C05448=1086.247,247.212,-78.817,176.012,22.627,153.611
C05449=1086.241,246.963,-78.790,176.009,22.624,153.611
C05450=1086.236,246.714,-78.763,176.007,22.621,153.611
C05451=1086.230,246.466,-78.736,176.004,22.619,153.611
C05452=1086.224,246.217,-78.710,176.002,22.616,153.610
C05453=1086.218,245.969,-78.683,175.999,22.613,153.610
C05454=1086.213,245.720,-78.656,175.996,22.610,153.610
C05455=1086.207,245.472,-78.629,175.994,22.607,153.610
C05456=1086.202,245.224,-78.603,175.991,22.604,153.610
C05457=1086.196,244.975,-78.576,175.988,22.602,153.609
C05458=1086.191,244.727,-78.549,175.985,22.598,153.609
C05459=1086.184,244.478,-78.522,175.982,22.596,153.609
C05460=1086.179,244.229,-78.495,175.980,22.593,153.608
C05461=1086.173,243.981,-78.468,175.977,22.590,153.608
C05462=1086.168,243.732,-78.441,175.974,22.587,153.608
C05463=1086.162,243.483,-78.415,175.972,22.584,153.608
C05464=1086.157,243.235,-78.389,175.969,22.581,153.608
C05465=1086.151,242.986,-78.362,175.967,22.578,153.607
C05466=1086.145,242.738,-78.335,175.964,22.576,153.607
C05467=1086.139,242.490,-78.309,175.961,22.573,153.607
C05468=1086.134,242.241,-78.282,175.958,22.570,153.607
C05469=1086.129,241.992,-78.255,175.955,22.567,153.607
C05470=1086.123,241.744,-78.229,175.953,22.564,153.606
C05471=1086.117,241.495,-78.202,175.950,22.561,153.606
C05472=1086.111,241.247,-78.176,175.947,22.558,153.606
C05473=1086.106,240.999,-78.149,175.945,22.556,153.606
C05474=1086.100,240.750,-78.123,175.942,22.553,153.605
C05475=1086.094,240.501,-78.096,175.939,22.550,153.605
C05476=1086.089,240.253,-78.070,175.936,22.547,153.605
C05477=1086.083,240.004,-78.044,175.934,22.544,153.605
C05478=1086.077,239.756,-78.017,175.931,22.542,153.604
C05479=1086.072,239.507,-77.990,175.928,22.538,153.604
C05480=1086.066,239.258,-77.964,175.926,22.536,153.604
C05481=1086.060,239.010,-77.938,175.923,22.533,153.604
C05482=1086.055,238.762,-77.911,175.921,22.530,153.604
C05483=1086.049,238.513,-77.885,175.918,22.527,153.603
C05484=1086.043,238.264,-77.859,175.915,22.525,153.603
C05485=1086.038,238.015,-77.833,175.912,22.522,153.603
C05486=1086.032,237.767,-77.806,175.909,22.519,153.603
C05487=1086.026,237.519,-77.779,175.907,22.516,153.602
C05488=1086.020,237.270,-77.754,175.904,22.513,153.602
C05489=1086.014,237.022,-77.727,175.902,22.511,153.602
C05490=1086.009,236.773,-77.701,175.899,22.507,153.602
C05491=1086.000,236.389,-77.661,175.895,22.503,153.601
C05492=1085.992,236.005,-77.620,175.891,22.498,153.601
C05493=1085.983,235.620,-77.580,175.887,22.495,153.601
C05494=1085.975,235.237,-77.539,175.882,22.490,153.601
C05495=1085.969,234.988,-77.513,175.880,22.487,153.600
C05496=1085.963,234.740,-77.487,175.877,22.484,153.600
C05497=1085.958,234.491,-77.461,175.875,22.482,153.600
C05498=1085.952,234.242,-77.435,175.872,22.479,153.600
C05499=1085.946,233.994,-77.409,175.869,22.476,153.599
C05500=1085.941,233.745,-77.383,175.867,22.473,153.599
C05501=1085.935,233.497,-77.357,175.864,22.470,153.599
C05502=1085.930,233.248,-77.331,175.861,22.467,153.599
C05503=1085.924,232.999,-77.305,175.858,22.464,153.598
C05504=1085.918,232.751,-77.279,175.856,22.462,153.598
C05505=1085.912,232.502,-77.253,175.853,22.459,153.598
C05506=1085.908,232.254,-77.227,175.851,22.456,153.598
C05507=1085.902,232.005,-77.201,175.848,22.453,153.598
C05508=1085.896,231.757,-77.175,175.846,22.451,153.597
C05509=1085.890,231.508,-77.149,175.843,22.447,153.597
C05510=1085.885,231.259,-77.123,175.840,22.445,153.597
C05511=1085.879,231.010,-77.097,175.837,22.442,153.597
C05512=1085.873,230.762,-77.072,175.835,22.440,153.596
C05513=1085.868,230.513,-77.046,175.832,22.436,153.596
C05514=1085.862,230.264,-77.020,175.829,22.434,153.596
C05515=1085.856,230.016,-76.994,175.827,22.431,153.596
C05516=1085.851,229.767,-76.969,175.824,22.428,153.596
C05517=1085.846,229.518,-76.943,175.822,22.425,153.595
C05518=1085.839,229.270,-76.917,175.819,22.422,153.595
C05519=1085.834,229.021,-76.891,175.816,22.420,153.595
C05520=1085.828,228.773,-76.866,175.813,22.417,153.595
C05521=1085.822,228.524,-76.840,175.811,22.414,153.594
C05522=1085.817,228.276,-76.815,175.808,22.411,153.594
C05523=1085.811,228.027,-76.789,175.806,22.408,153.594
C05524=1085.806,227.778,-76.763,175.803,22.406,153.594
C05525=1085.799,227.529,-76.738,175.801,22.403,153.594
C05526=1085.795,227.281,-76.712,175.798,22.400,153.594
C05527=1085.788,227.032,-76.687,175.795,22.397,153.593
C05528=1085.783,226.783,-76.661,175.792,22.395,153.593
C05529=1085.777,226.535,-76.635,175.790,22.392,153.593
C05530=1085.772,226.286,-76.610,175.787,22.389,153.593
C05531=1085.766,226.038,-76.584,175.785,22.386,153.592
C05532=1085.760,225.789,-76.559,175.782,22.383,153.592
C05533=1085.754,225.541,-76.534,175.780,22.381,153.592
C05534=1085.749,225.292,-76.508,175.777,22.378,153.592
C05535=1085.743,225.043,-76.482,175.775,22.375,153.591
C05536=1085.737,224.794,-76.456,175.772,22.373,153.591
C05537=1085.732,224.546,-76.431,175.769,22.369,153.591
C05538=1085.726,224.297,-76.405,175.767,22.367,153.591
C05539=1085.720,224.048,-76.380,175.764,22.364,153.591
C05540=1085.716,223.800,-76.355,175.762,22.362,153.590
C05541=1085.709,223.551,-76.330,175.759,22.358,153.590
C05542=1085.704,223.302,-76.304,175.757,22.356,153.590
C05543=1085.695,222.910,-76.264,175.752,22.351,153.590
C05544=1085.686,222.517,-76.225,175.748,22.347,153.589
C05545=1085.677,222.124,-76.184,175.744,22.342,153.589
C05546=1085.669,221.732,-76.144,175.740,22.338,153.589
C05547=1085.663,221.483,-76.119,175.737,22.335,153.588
C05548=1085.657,221.235,-76.094,175.735,22.333,153.588
C05549=1085.651,220.986,-76.069,175.732,22.329,153.588
C05550=1085.646,220.737,-76.043,175.730,22.327,153.588
C05551=1085.640,220.488,-76.019,175.727,22.324,153.588
C05552=1085.634,220.240,-75.994,175.724,22.321,153.587
C05553=1085.629,219.992,-75.969,175.722,22.319,153.587
C05554=1085.623,219.742,-75.943,175.719,22.316,153.587
C05555=1085.617,219.493,-75.918,175.717,22.314,153.587
C05556=1085.612,219.246,-75.893,175.714,22.310,153.587
C05557=1085.606,218.996,-75.868,175.712,22.308,153.586
C05558=1085.601,218.748,-75.843,175.709,22.305,153.586
C05559=1085.595,218.499,-75.818,175.706,22.302,153.586
C05560=1085.589,218.250,-75.793,175.704,22.299,153.586
C05561=1085.583,218.002,-75.768,175.701,22.297,153.586
C05562=1085.578,217.752,-75.743,175.699,22.294,153.585
C05563=1085.572,217.504,-75.718,175.696,22.291,153.585
C05564=1085.567,217.255,-75.693,175.694,22.288,153.585
C05565=1085.561,217.007,-75.668,175.691,22.286,153.585
C05566=1085.555,216.758,-75.644,175.689,22.283,153.584
C05567=1085.550,216.510,-75.618,175.686,22.280,153.584
C05568=1085.544,216.260,-75.593,175.684,22.277,153.584
C05569=1085.539,216.012,-75.568,175.681,22.275,153.584
C05570=1085.533,215.763,-75.544,175.678,22.272,153.584
C05571=1085.527,215.515,-75.519,175.676,22.269,153.583
C05572=1085.521,215.266,-75.494,175.673,22.266,153.583
C05573=1085.516,215.018,-75.469,175.671,22.264,153.583
C05574=1085.510,214.768,-75.444,175.668,22.260,153.583
C05575=1085.505,214.520,-75.420,175.666,22.258,153.583
C05576=1085.499,214.271,-75.394,175.663,22.255,153.582
C05577=1085.494,214.022,-75.370,175.660,22.252,153.582
C05578=1085.487,213.774,-75.345,175.658,22.250,153.582
C05579=1085.483,213.525,-75.320,175.655,22.247,153.582
C05580=1085.477,213.276,-75.295,175.653,22.244,153.581
C05581=1085.471,213.028,-75.270,175.650,22.241,153.581
C05582=1085.465,212.778,-75.246,175.648,22.238,153.581
C05583=1085.460,212.530,-75.222,175.646,22.236,153.581
C05584=1085.455,212.281,-75.197,175.643,22.233,153.581
C05585=1085.449,212.032,-75.172,175.640,22.231,153.580
C05586=1085.443,211.784,-75.148,175.637,22.227,153.580
C05587=1085.437,211.535,-75.123,175.635,22.225,153.580
C05588=1085.432,211.286,-75.099,175.633,22.222,153.580
C05589=1085.426,211.037,-75.073,175.630,22.219,153.580
C05590=1085.421,210.789,-75.049,175.628,22.216,153.579
C05591=1085.415,210.540,-75.025,175.625,22.214,153.579
C05592=1085.409,210.291,-75.000,175.622,22.211,153.579
C05593=1085.404,210.042,-74.976,175.620,22.209,153.579
C05594=1085.398,209.794,-74.951,175.617,22.206,153.579
C05595=1085.388,209.405,-74.913,175.614,22.202,153.578
C05596=1085.380,209.017,-74.875,175.610,22.197,153.578
C05597=1085.372,208.628,-74.837,175.605,22.193,153.578
C05598=1085.363,208.239,-74.799,175.602,22.188,153.577
C05599=1085.339,207.211,-74.700,175.519,22.146,153.580
C05600=1085.334,206.963,-74.676,175.517,22.144,153.580
C05601=1085.329,206.714,-74.652,175.514,22.142,153.580
C05602=1085.322,206.465,-74.628,175.511,22.140,153.580
C05603=1085.317,206.216,-74.604,175.509,22.138,153.580
C05604=1085.312,205.967,-74.580,175.506,22.136,153.580
C05605=1085.306,205.718,-74.557,175.504,22.135,153.580
C05606=1085.301,205.470,-74.533,175.501,22.133,153.580
C05607=1085.295,205.221,-74.508,175.498,22.131,153.580
C05608=1085.289,204.972,-74.485,175.495,22.129,153.580
C05609=1085.284,204.723,-74.461,175.493,22.127,153.580
C05610=1085.278,204.475,-74.437,175.490,22.125,153.580
C05611=1085.273,204.226,-74.414,175.488,22.123,153.580
C05612=1085.267,203.977,-74.389,175.485,22.122,153.580
C05613=1085.262,203.728,-74.366,175.483,22.120,153.580
C05614=1085.256,203.480,-74.342,175.479,22.118,153.580
C05615=1085.251,203.230,-74.317,175.477,22.116,153.580
C05616=1085.245,202.981,-74.295,175.475,22.114,153.580
C05617=1085.239,202.733,-74.270,175.472,22.112,153.580
C05618=1085.234,202.484,-74.247,175.470,22.111,153.580
C05619=1085.228,202.235,-74.223,175.467,22.109,153.580
C05620=1085.223,201.986,-74.200,175.465,22.107,153.580
C05621=1085.217,201.738,-74.176,175.462,22.106,153.580
C05622=1085.211,201.488,-74.153,175.459,22.103,153.580
C05623=1085.205,201.240,-74.129,175.456,22.102,153.581
C05624=1085.199,200.991,-74.106,175.454,22.100,153.581
C05625=1085.194,200.742,-74.082,175.451,22.098,153.580
C05626=1085.188,200.494,-74.059,175.449,22.096,153.580
C05627=1085.183,200.245,-74.034,175.446,22.095,153.581
C05628=1085.177,199.996,-74.012,175.444,22.093,153.581
C05629=1085.171,199.746,-73.988,175.441,22.091,153.581
C05630=1085.166,199.498,-73.964,175.439,22.090,153.581
C05631=1085.160,199.249,-73.941,175.435,22.088,153.581
C05632=1085.154,199.001,-73.917,175.433,22.086,153.581
C05633=1085.149,198.752,-73.894,175.430,22.084,153.581
C05634=1085.143,198.503,-73.871,175.428,22.082,153.581
C05635=1085.137,198.254,-73.847,175.426,22.081,153.581
C05636=1085.132,198.005,-73.824,175.423,22.079,153.581
C05637=1085.126,197.756,-73.801,175.420,22.077,153.581
C05638=1085.120,197.508,-73.777,175.418,22.076,153.581
C05639=1085.115,197.259,-73.754,175.416,22.074,153.581
C05640=1085.110,197.010,-73.731,175.413,22.072,153.581
C05641=1085.104,196.762,-73.707,175.410,22.070,153.581
C05642=1085.098,196.513,-73.684,175.407,22.068,153.581
C05643=1085.093,196.263,-73.660,175.405,22.066,153.581
C05644=1085.087,196.015,-73.638,175.402,22.065,153.581
C05645=1085.081,195.765,-73.614,175.400,22.063,153.581
C05646=1085.076,195.516,-73.590,175.397,22.061,153.581
C05647=1085.070,195.267,-73.567,175.395,22.060,153.581
C05648=1085.064,195.019,-73.544,175.392,22.058,153.581
C05649=1085.058,194.770,-73.521,175.390,22.056,153.581
C05650=1085.054,194.521,-73.498,175.387,22.054,153.581
C05651=1085.048,194.273,-73.474,175.385,22.052,153.581
C05652=1085.042,194.024,-73.451,175.382,22.050,153.581
C05653=1085.036,193.775,-73.428,175.380,22.049,153.581
C05654=1085.031,193.526,-73.405,175.377,22.047,153.581
C05655=1085.026,193.277,-73.382,175.375,22.045,153.581
C05656=1085.020,193.028,-73.359,175.372,22.043,153.581
C05657=1085.014,192.779,-73.336,175.369,22.041,153.581
C05658=1085.009,192.531,-73.312,175.367,22.039,153.581
C05659=1085.003,192.282,-73.289,175.364,22.038,153.581
C05660=1084.997,192.003,-73.264,175.362,22.036,153.581
C05661=1084.990,191.725,-73.238,175.358,22.033,153.581
C05662=1084.985,191.447,-73.211,175.356,22.032,153.581
C05663=1084.978,191.168,-73.187,175.354,22.030,153.581
C05664=1084.973,190.919,-73.163,175.351,22.028,153.581
C05665=1084.968,190.670,-73.140,175.349,22.026,153.581
C05666=1084.962,190.421,-73.117,175.346,22.024,153.581
C05667=1084.956,190.172,-73.094,175.344,22.022,153.581
C05668=1084.950,189.923,-73.071,175.340,22.021,153.581
C05669=1084.946,189.675,-73.048,175.338,22.019,153.581
C05670=1084.940,189.426,-73.025,175.335,22.017,153.581
C05671=1084.935,189.177,-73.002,175.333,22.015,153.581
C05672=1084.929,188.928,-72.979,175.330,22.013,153.581
C05673=1084.923,188.679,-72.956,175.328,22.011,153.581
C05674=1084.917,188.430,-72.933,175.326,22.010,153.581
C05675=1084.913,188.182,-72.910,175.323,22.008,153.581
C05676=1084.907,187.933,-72.887,175.321,22.006,153.581
C05677=1084.902,187.684,-72.864,175.318,22.004,153.581
C05678=1084.896,187.435,-72.841,175.316,22.002,153.581
C05679=1084.890,187.186,-72.819,175.313,22.000,153.581
C05680=1084.885,186.937,-72.796,175.311,21.999,153.581
C05681=1084.879,186.689,-72.774,175.308,21.997,153.581
C05682=1084.874,186.439,-72.750,175.306,21.995,153.581
C05683=1084.869,186.190,-72.727,175.304,21.993,153.581
C05684=1084.863,185.941,-72.705,175.301,21.991,153.581
C05685=1084.858,185.693,-72.682,175.299,21.989,153.580
C05686=1084.852,185.444,-72.659,175.296,21.988,153.580
C05687=1084.847,185.195,-72.636,175.294,21.986,153.580
C05688=1084.841,184.946,-72.613,175.291,21.984,153.580
C05689=1084.836,184.697,-72.591,175.289,21.982,153.580
C05690=1084.830,184.448,-72.568,175.286,21.981,153.581
C05691=1084.824,184.200,-72.546,175.284,21.979,153.581
C05692=1084.818,183.951,-72.523,175.281,21.977,153.581
C05693=1084.813,183.701,-72.501,175.279,21.975,153.580
C05694=1084.807,183.452,-72.478,175.276,21.974,153.581
C05695=1084.801,183.204,-72.456,175.274,21.972,153.581
C05696=1084.795,182.954,-72.434,175.271,21.970,153.581
C05697=1084.789,182.705,-72.411,175.269,21.968,153.581
C05698=1084.784,182.457,-72.388,175.266,21.966,153.581
C05699=1084.778,182.208,-72.366,175.264,21.965,153.581
C05700=1084.772,181.959,-72.343,175.261,21.963,153.581
C05701=1084.767,181.710,-72.321,175.259,21.961,153.581
C05702=1084.761,181.461,-72.298,175.257,21.960,153.581
C05703=1084.755,181.212,-72.276,175.255,21.958,153.581
C05704=1084.750,180.963,-72.254,175.252,21.957,153.581
C05705=1084.744,180.714,-72.231,175.250,21.955,153.581
C05706=1084.739,180.465,-72.209,175.247,21.953,153.581
C05707=1084.732,180.216,-72.187,175.245,21.951,153.581
C05708=1084.727,179.967,-72.164,175.243,21.950,153.581
C05709=1084.722,179.719,-72.142,175.240,21.948,153.581
C05710=1084.715,179.470,-72.119,175.238,21.946,153.581
C05711=1084.710,179.221,-72.097,175.235,21.944,153.581
C05712=1084.704,178.972,-72.074,175.233,21.943,153.581
C05713=1084.699,178.723,-72.053,175.230,21.941,153.581
C05714=1084.693,178.474,-72.030,175.228,21.939,153.581
C05715=1084.687,178.225,-72.008,175.225,21.937,153.581
C05716=1084.681,177.975,-71.986,175.223,21.935,153.581
C05717=1084.676,177.727,-71.964,175.220,21.933,153.581
C05718=1084.671,177.478,-71.941,175.218,21.932,153.581
C05719=1084.664,177.229,-71.919,175.215,21.930,153.581
C05720=1084.659,176.980,-71.897,175.213,21.928,153.581
C05721=1084.654,176.731,-71.874,175.210,21.927,153.581
C05722=1084.648,176.482,-71.853,175.209,21.925,153.581
C05723=1084.642,176.233,-71.830,175.206,21.923,153.581
C05724=1084.636,175.954,-71.806,175.203,21.921,153.581
C05725=1084.630,175.676,-71.781,175.201,21.919,153.581
C05726=1084.623,175.398,-71.756,175.198,21.917,153.581
C05727=1084.617,175.119,-71.731,175.196,21.916,153.581
C05728=1084.612,174.870,-71.709,175.193,21.914,153.581
C05729=1084.606,174.620,-71.687,175.191,21.912,153.581
C05730=1084.600,174.372,-71.665,175.188,21.910,153.581
C05731=1084.595,174.123,-71.642,175.186,21.908,153.581
C05732=1084.589,173.874,-71.621,175.183,21.906,153.581
C05733=1084.584,173.625,-71.599,175.181,21.904,153.580
C05734=1084.578,173.376,-71.576,175.179,21.903,153.580
C05735=1084.573,173.127,-71.555,175.176,21.901,153.580
C05736=1084.567,172.878,-71.532,175.174,21.899,153.580
C05737=1084.561,172.629,-71.511,175.171,21.897,153.580
C05738=1084.556,172.380,-71.488,175.169,21.895,153.580
C05739=1084.550,172.131,-71.467,175.167,21.894,153.580
C05740=1084.545,171.882,-71.445,175.165,21.892,153.580
C05741=1084.539,171.633,-71.423,175.162,21.890,153.580
C05742=1084.533,171.384,-71.401,175.160,21.888,153.580
C05743=1084.528,171.136,-71.378,175.158,21.886,153.580
C05744=1084.522,170.886,-71.357,175.155,21.885,153.580
C05745=1084.517,170.637,-71.335,175.153,21.883,153.580
C05746=1084.511,170.388,-71.313,175.150,21.881,153.580
C05747=1084.506,170.139,-71.291,175.148,21.879,153.580
C05748=1084.500,169.890,-71.270,175.146,21.878,153.580
C05749=1084.495,169.641,-71.247,175.144,21.876,153.580
C05750=1084.489,169.392,-71.226,175.141,21.874,153.580
C05751=1084.483,169.143,-71.203,175.139,21.872,153.580
C05752=1084.478,168.895,-71.181,175.136,21.870,153.580
C05753=1084.472,168.645,-71.160,175.134,21.868,153.580
C05754=1084.467,168.397,-71.138,175.132,21.866,153.580
C05755=1084.461,168.147,-71.116,175.129,21.864,153.580
C05756=1084.457,167.898,-71.094,175.127,21.862,153.580
C05757=1084.450,167.649,-71.073,175.125,21.861,153.580
C05758=1084.446,167.400,-71.051,175.123,21.859,153.580
C05759=1084.439,167.151,-71.029,175.120,21.857,153.580
C05760=1084.435,166.902,-71.007,175.118,21.855,153.580
C05761=1084.428,166.653,-70.986,175.116,21.854,153.580
C05762=1084.424,166.404,-70.964,175.113,21.852,153.580
C05763=1084.418,166.156,-70.943,175.111,21.849,153.580
C05764=1084.412,165.907,-70.921,175.109,21.848,153.580
C05765=1084.407,165.658,-70.899,175.107,21.846,153.580
C05766=1084.401,165.409,-70.877,175.104,21.844,153.580
C05767=1084.396,165.160,-70.856,175.102,21.842,153.580
C05768=1084.390,164.910,-70.835,175.100,21.841,153.580
C05769=1084.385,164.661,-70.813,175.097,21.839,153.580
C05770=1084.380,164.413,-70.792,175.095,21.836,153.579
C05771=1084.374,164.163,-70.769,175.093,21.835,153.579
C05772=1084.369,163.915,-70.748,175.091,21.833,153.579
C05773=1084.363,163.665,-70.726,175.088,21.831,153.579
C05774=1084.358,163.417,-70.705,175.086,21.830,153.579
C05775=1084.353,163.168,-70.684,175.084,21.828,153.579
C05776=1084.347,162.918,-70.662,175.081,21.825,153.579
C05777=1084.342,162.670,-70.641,175.079,21.823,153.579
C05778=1084.336,162.420,-70.618,175.077,21.822,153.579
C05779=1084.331,162.172,-70.597,175.075,21.820,153.579
C05780=1084.326,161.923,-70.575,175.072,21.818,153.579
C05781=1084.320,161.673,-70.554,175.070,21.816,153.579
C05782=1084.314,161.424,-70.533,175.068,21.814,153.579
C05783=1084.308,161.175,-70.511,175.065,21.812,153.579
C05784=1084.303,160.926,-70.489,175.064,21.811,153.579
C05785=1084.298,160.677,-70.469,175.061,21.809,153.579
C05786=1084.292,160.428,-70.447,175.059,21.807,153.579
C05787=1084.286,160.180,-70.426,175.056,21.805,153.579
C05788=1084.280,159.901,-70.402,175.054,21.804,153.579
C05789=1084.273,159.621,-70.378,175.052,21.801,153.579
C05790=1084.267,159.342,-70.354,175.049,21.799,153.579
C05791=1084.261,159.062,-70.331,175.046,21.797,153.579
C05792=1084.256,158.814,-70.309,175.044,21.796,153.579
C05793=1084.250,158.565,-70.288,175.042,21.794,153.579
C05794=1084.244,158.316,-70.267,175.040,21.792,153.579
C05795=1084.239,158.067,-70.246,175.037,21.790,153.579
C05796=1084.233,157.818,-70.224,175.035,21.788,153.578
C05797=1084.227,157.569,-70.204,175.033,21.786,153.578
C05798=1084.222,157.320,-70.182,175.031,21.784,153.578
C05799=1084.217,157.070,-70.161,175.028,21.783,153.578
C05800=1084.211,156.822,-70.140,175.026,21.781,153.578
C05801=1084.206,156.573,-70.118,175.024,21.779,153.578
C05802=1084.200,156.323,-70.097,175.022,21.777,153.578
C05803=1084.194,156.075,-70.076,175.020,21.775,153.578
C05804=1084.189,155.826,-70.056,175.017,21.773,153.578
C05805=1084.183,155.577,-70.034,175.015,21.771,153.578
C05806=1084.178,155.327,-70.013,175.012,21.770,153.578
C05807=1084.172,155.079,-69.992,175.011,21.768,153.578
C05808=1084.166,154.829,-69.971,175.008,21.766,153.578
C05809=1084.161,154.581,-69.950,175.006,21.764,153.578
C05810=1084.155,154.331,-69.929,175.004,21.763,153.578
C05811=1084.149,154.082,-69.908,175.001,21.760,153.578
C05812=1084.144,153.833,-69.887,175.000,21.759,153.578
C05813=1084.138,153.585,-69.866,174.997,21.757,153.578
C05814=1084.132,153.335,-69.845,174.995,21.755,153.578
C05815=1084.127,153.086,-69.824,174.993,21.753,153.578
C05816=1084.122,152.837,-69.803,174.991,21.752,153.578
C05817=1084.116,152.587,-69.782,174.989,21.750,153.578
C05818=1084.110,152.339,-69.761,174.986,21.748,153.578
C05819=1084.105,152.090,-69.740,174.984,21.746,153.578
C05820=1084.099,151.841,-69.719,174.981,21.744,153.578
C05821=1084.094,151.591,-69.698,174.980,21.743,153.578
C05822=1084.088,151.342,-69.678,174.978,21.740,153.577
C05823=1084.082,151.094,-69.657,174.975,21.738,153.577
C05824=1084.076,150.844,-69.636,174.973,21.737,153.577
C05825=1084.071,150.595,-69.616,174.971,21.735,153.577
C05826=1084.065,150.347,-69.594,174.969,21.733,153.577
C05827=1084.060,150.097,-69.574,174.967,21.731,153.577
C05828=1084.054,149.848,-69.553,174.964,21.729,153.577
C05829=1084.049,149.599,-69.532,174.963,21.728,153.577
C05830=1084.043,149.350,-69.511,174.960,21.726,153.577
C05831=1084.038,149.101,-69.490,174.958,21.723,153.577
C05832=1084.032,148.851,-69.470,174.955,21.722,153.577
C05833=1084.026,148.603,-69.449,174.954,21.720,153.577
C05834=1084.021,148.354,-69.428,174.951,21.718,153.577
C05835=1084.015,148.105,-69.408,174.949,21.716,153.577
C05836=1084.010,147.856,-69.387,174.947,21.714,153.577
C05837=1084.003,147.607,-69.366,174.945,21.713,153.577
C05838=1083.998,147.357,-69.346,174.943,21.711,153.577
C05839=1083.993,147.108,-69.325,174.940,21.709,153.577
C05840=1083.988,146.859,-69.305,174.938,21.707,153.577
C05841=1083.981,146.610,-69.284,174.937,21.705,153.576
C05842=1083.975,146.361,-69.263,174.934,21.703,153.576
C05843=1083.970,146.112,-69.242,174.932,21.701,153.576
C05844=1083.965,145.863,-69.222,174.929,21.700,153.576
C05845=1083.959,145.614,-69.202,174.928,21.698,153.576
C05846=1083.953,145.364,-69.181,174.925,21.696,153.576
C05847=1083.948,145.115,-69.160,174.923,21.694,153.576
C05848=1083.942,144.866,-69.140,174.921,21.692,153.576
C05849=1083.937,144.617,-69.120,174.919,21.690,153.576
C05850=1083.931,144.369,-69.099,174.917,21.688,153.576
C05851=1083.924,144.119,-69.078,174.914,21.687,153.576
C05852=1083.919,143.840,-69.055,174.912,21.685,153.576
C05853=1083.913,143.561,-69.032,174.910,21.682,153.576
C05854=1083.906,143.282,-69.010,174.907,21.680,153.576
C05855=1083.900,143.002,-68.987,174.905,21.678,153.576
C05856=1083.895,142.753,-68.966,174.903,21.676,153.576
C05857=1083.889,142.503,-68.945,174.901,21.675,153.576
C05858=1083.883,142.255,-68.926,174.899,21.672,153.576
C05859=1083.878,142.005,-68.905,174.896,21.671,153.576
C05860=1083.872,141.756,-68.884,174.894,21.669,153.576
C05861=1083.866,141.508,-68.864,174.893,21.667,153.575
C05862=1083.861,141.258,-68.844,174.890,21.665,153.575
C05863=1083.855,141.010,-68.824,174.888,21.663,153.575
C05864=1083.850,140.760,-68.803,174.886,21.661,153.575
C05865=1083.845,140.511,-68.783,174.884,21.659,153.575
C05866=1083.838,140.262,-68.762,174.882,21.657,153.575
C05867=1083.833,140.013,-68.742,174.879,21.655,153.575
C05868=1083.827,139.764,-68.722,174.878,21.654,153.575
C05869=1083.822,139.515,-68.701,174.875,21.652,153.575
C05870=1083.816,139.265,-68.682,174.873,21.649,153.575
C05871=1083.811,139.016,-68.662,174.872,21.648,153.575
C05872=1083.805,138.767,-68.641,174.869,21.646,153.575
C05873=1083.799,138.518,-68.621,174.867,21.644,153.575
C05874=1083.794,138.269,-68.601,174.865,21.642,153.575
C05875=1083.788,138.020,-68.581,174.863,21.641,153.575
C05876=1083.783,137.771,-68.560,174.861,21.638,153.574
C05877=1083.777,137.521,-68.540,174.858,21.636,153.574
C05878=1083.771,137.272,-68.520,174.857,21.635,153.574
C05879=1083.765,137.023,-68.500,174.854,21.633,153.574
C05880=1083.759,136.774,-68.480,174.852,21.631,153.574
C05881=1083.754,136.525,-68.459,174.850,21.629,153.574
C05882=1083.748,136.276,-68.440,174.848,21.627,153.574
C05883=1083.743,136.027,-68.420,174.846,21.625,153.574
C05884=1083.737,135.778,-68.400,174.844,21.624,153.574
C05885=1083.732,135.529,-68.379,174.842,21.621,153.574
C05886=1083.726,135.279,-68.360,174.840,21.619,153.574
C05887=1083.720,135.030,-68.340,174.838,21.618,153.574
C05888=1083.715,134.781,-68.319,174.836,21.616,153.574
C05889=1083.709,134.533,-68.299,174.833,21.614,153.574
C05890=1083.704,134.283,-68.280,174.832,21.612,153.573
C05891=1083.698,134.034,-68.260,174.830,21.610,153.573
C05892=1083.693,133.785,-68.239,174.827,21.608,153.573
C05893=1083.687,133.535,-68.220,174.826,21.606,153.573
C05894=1083.681,133.287,-68.200,174.823,21.604,153.573
C05895=1083.676,133.038,-68.179,174.821,21.602,153.573
C05896=1083.670,132.788,-68.160,174.820,21.601,153.573
C05897=1083.665,132.539,-68.139,174.817,21.599,153.573
C05898=1083.659,132.290,-68.120,174.815,21.596,153.573
C05899=1083.653,132.041,-68.100,174.813,21.595,153.573
C05900=1083.647,131.792,-68.080,174.811,21.593,153.573
C05901=1083.642,131.542,-68.060,174.809,21.591,153.573
C05902=1083.636,131.293,-68.041,174.807,21.589,153.573
C05903=1083.631,131.044,-68.021,174.805,21.587,153.572
C05904=1083.625,130.795,-68.001,174.803,21.585,153.572
C05905=1083.619,130.546,-67.981,174.801,21.584,153.572
C05906=1083.614,130.297,-67.962,174.799,21.581,153.572
C05907=1083.608,130.048,-67.942,174.796,21.579,153.572
C05908=1083.602,129.798,-67.922,174.795,21.578,153.572
C05909=1083.596,129.549,-67.902,174.793,21.576,153.572
C05910=1083.590,129.300,-67.883,174.790,21.574,153.572
C05911=1083.584,129.051,-67.863,174.789,21.572,153.572
C05912=1083.579,128.801,-67.843,174.786,21.570,153.572
C05913=1083.573,128.553,-67.823,174.784,21.568,153.572
C05914=1083.568,128.303,-67.804,174.783,21.566,153.572
C05915=1083.562,128.054,-67.784,174.780,21.564,153.572
C05916=1083.556,127.774,-67.762,174.778,21.562,153.572
C05917=1083.548,127.495,-67.740,174.776,21.560,153.572
C05918=1083.543,127.216,-67.718,174.773,21.558,153.571
C05919=1083.536,126.937,-67.697,174.771,21.555,153.571
C05920=1083.531,126.687,-67.676,174.770,21.554,153.571
C05921=1083.525,126.438,-67.657,174.767,21.552,153.571
C05922=1083.519,126.189,-67.637,174.765,21.550,153.571
C05923=1083.513,125.940,-67.618,174.763,21.548,153.571
C05924=1083.508,125.690,-67.599,174.761,21.546,153.571
C05925=1083.502,125.442,-67.579,174.760,21.545,153.571
C05926=1083.497,125.193,-67.560,174.757,21.542,153.571
C05927=1083.491,124.943,-67.540,174.755,21.540,153.571
C05928=1083.485,124.695,-67.520,174.754,21.538,153.571
C05929=1083.480,124.445,-67.501,174.751,21.536,153.571
C05930=1083.474,124.195,-67.481,174.749,21.534,153.570
C05931=1083.468,123.947,-67.461,174.747,21.533,153.570
C05932=1083.463,123.697,-67.442,174.745,21.530,153.570
C05933=1083.457,123.448,-67.423,174.744,21.529,153.570
C05934=1083.452,123.200,-67.403,174.741,21.527,153.570
C05935=1083.446,122.950,-67.384,174.739,21.525,153.570
C05936=1083.440,122.701,-67.365,174.738,21.523,153.570
C05937=1083.435,122.451,-67.346,174.735,21.521,153.570
C05938=1083.429,122.203,-67.326,174.733,21.518,153.570
C05939=1083.423,121.953,-67.306,174.731,21.517,153.570
C05940=1083.418,121.704,-67.288,174.729,21.515,153.570
C05941=1083.412,121.455,-67.268,174.728,21.513,153.569
C05942=1083.406,121.205,-67.249,174.725,21.511,153.569
C05943=1083.400,120.957,-67.229,174.723,21.509,153.569
C05944=1083.395,120.707,-67.209,174.722,21.507,153.569
C05945=1083.390,120.458,-67.190,174.719,21.505,153.569
C05946=1083.385,120.209,-67.171,174.718,21.503,153.569
C05947=1083.379,119.959,-67.152,174.716,21.501,153.569
C05948=1083.373,119.711,-67.132,174.713,21.499,153.569
C05949=1083.367,119.461,-67.113,174.712,21.497,153.569
C05950=1083.362,119.212,-67.094,174.710,21.495,153.568
C05951=1083.357,118.963,-67.075,174.708,21.493,153.568
C05952=1083.351,118.713,-67.055,174.706,21.491,153.568
C05953=1083.345,118.464,-67.036,174.704,21.489,153.568
C05954=1083.340,118.215,-67.017,174.702,21.487,153.568
C05955=1083.334,117.966,-66.998,174.700,21.485,153.568
C05956=1083.329,117.716,-66.979,174.699,21.483,153.568
C05957=1083.323,117.468,-66.959,174.696,21.481,153.568
C05958=1083.318,117.219,-66.940,174.694,21.479,153.568
C05959=1083.312,116.969,-66.921,174.693,21.477,153.567
C05960=1083.306,116.720,-66.901,174.690,21.475,153.567
C05961=1083.301,116.471,-66.883,174.689,21.473,153.567
C05962=1083.295,116.222,-66.863,174.687,21.470,153.567
C05963=1083.290,115.972,-66.844,174.684,21.469,153.567
C05964=1083.284,115.723,-66.825,174.683,21.467,153.567
C05965=1083.279,115.474,-66.806,174.681,21.464,153.567
C05966=1083.273,115.225,-66.787,174.679,21.463,153.567
C05967=1083.268,114.975,-66.767,174.677,21.461,153.567
C05968=1083.262,114.727,-66.749,174.675,21.459,153.566
C05969=1083.256,114.478,-66.730,174.673,21.456,153.566
C05970=1083.250,114.228,-66.711,174.671,21.454,153.566
C05971=1083.245,113.979,-66.692,174.669,21.452,153.566
C05972=1083.240,113.729,-66.673,174.667,21.451,153.566
C05973=1083.234,113.480,-66.654,174.666,21.449,153.566
C05974=1083.228,113.231,-66.635,174.663,21.446,153.566
C05975=1083.223,112.982,-66.616,174.662,21.445,153.566
C05976=1083.217,112.733,-66.597,174.660,21.442,153.566
C05977=1083.211,112.483,-66.578,174.658,21.440,153.565
C05978=1083.206,112.235,-66.560,174.656,21.439,153.565
C05979=1083.200,111.985,-66.540,174.654,21.436,153.565
C05980=1083.195,111.754,-66.523,174.652,21.435,153.565
C05981=1083.190,111.524,-66.505,174.651,21.433,153.565
C05982=1083.184,111.293,-66.488,174.649,21.430,153.565
C05983=1083.179,111.062,-66.471,174.647,21.429,153.565
C05984=1083.174,110.832,-66.453,174.645,21.427,153.565
C05985=1083.169,110.601,-66.436,174.643,21.425,153.565
C05986=1083.163,110.370,-66.419,174.642,21.423,153.565
C05987=1083.158,110.141,-66.401,174.640,21.421,153.565
C05988=1083.152,109.891,-66.382,174.638,21.420,153.564
C05989=1083.147,109.641,-66.364,174.636,21.418,153.564
C05990=1083.140,109.392,-66.345,174.634,21.416,153.564
C05991=1083.135,109.143,-66.326,174.632,21.413,153.564
C05992=1083.130,108.894,-66.307,174.631,21.412,153.564
C05993=1083.123,108.645,-66.288,174.628,21.410,153.564
C05994=1083.118,108.396,-66.270,174.626,21.407,153.564
C05995=1083.113,108.146,-66.251,174.625,21.406,153.564
C05996=1083.107,107.898,-66.233,174.623,21.403,153.564
C05997=1083.101,107.648,-66.214,174.621,21.401,153.563
C05998=1083.095,107.399,-66.195,174.619,21.400,153.563
C05999=1083.090,107.150,-66.177,174.617,21.398,153.563
C06000=1083.084,106.900,-66.157,174.615,21.395,153.563
C06001=1083.078,106.651,-66.139,174.614,21.393,153.563
C06002=1083.073,106.402,-66.120,174.611,21.391,153.563
C06003=1083.067,106.153,-66.102,174.610,21.389,153.563
C06004=1083.062,105.903,-66.084,174.608,21.387,153.563
C06005=1083.056,105.654,-66.064,174.606,21.385,153.562
C06006=1083.050,105.404,-66.046,174.604,21.383,153.562
C06007=1083.045,105.156,-66.028,174.602,21.381,153.562
C06008=1083.038,104.906,-66.009,174.601,21.379,153.562
C06009=1083.034,104.657,-65.991,174.598,21.377,153.562
C06010=1083.027,104.408,-65.972,174.597,21.375,153.562
C06011=1083.022,104.159,-65.953,174.595,21.373,153.562
C06012=1083.017,103.909,-65.935,174.593,21.371,153.562
C06013=1083.010,103.660,-65.916,174.591,21.368,153.561
C06014=1083.006,103.411,-65.898,174.590,21.367,153.561
C06015=1082.999,103.162,-65.879,174.587,21.365,153.561
C06016=1082.993,102.845,-65.856,174.585,21.362,153.561
C06017=1082.986,102.528,-65.833,174.583,21.359,153.561
C06018=1082.978,102.212,-65.809,174.580,21.356,153.561
C06019=1082.971,101.895,-65.785,174.578,21.354,153.561
C06020=1082.966,101.645,-65.767,174.576,21.352,153.560
C06021=1082.960,101.396,-65.749,174.574,21.350,153.560
C06022=1082.955,101.147,-65.730,174.573,21.348,153.560
C06023=1082.949,100.898,-65.712,174.571,21.345,153.560
C06024=1082.942,100.648,-65.694,174.569,21.344,153.560
C06025=1082.937,100.399,-65.675,174.567,21.342,153.560
C06026=1082.931,100.150,-65.657,174.566,21.340,153.560
C06027=1082.925,99.901,-65.639,174.563,21.337,153.559
C06028=1082.920,99.651,-65.620,174.562,21.336,153.559
C06029=1082.915,99.402,-65.603,174.560,21.333,153.559
C06030=1082.908,99.153,-65.584,174.558,21.332,153.559
C06031=1082.903,98.904,-65.566,174.556,21.329,153.559
C06032=1082.897,98.655,-65.547,174.555,21.328,153.559
C06033=1082.891,98.405,-65.530,174.552,21.325,153.559
C06034=1082.886,98.155,-65.511,174.551,21.323,153.559
C06035=1082.880,97.907,-65.493,174.549,21.321,153.558
C06036=1082.874,97.657,-65.475,174.547,21.319,153.558
C06037=1082.869,97.407,-65.456,174.545,21.317,153.558
C06038=1082.863,97.159,-65.438,174.544,21.315,153.558
C06039=1082.857,96.910,-65.420,174.541,21.313,153.558
C06040=1082.852,96.660,-65.402,174.539,21.310,153.558
C06041=1082.846,96.411,-65.384,174.538,21.308,153.558
C06042=1082.840,96.162,-65.366,174.536,21.306,153.557
C06043=1082.835,95.912,-65.348,174.534,21.305,153.557
C06044=1082.828,95.634,-65.327,174.532,21.302,153.557
C06045=1082.822,95.353,-65.306,174.530,21.299,153.557
C06046=1082.815,95.074,-65.287,174.529,21.297,153.557
C06047=1082.809,94.795,-65.266,174.526,21.295,153.557
C06048=1082.804,94.545,-65.249,174.524,21.293,153.557
C06049=1082.797,94.296,-65.230,174.523,21.291,153.557
C06050=1082.792,94.047,-65.212,174.520,21.289,153.556
C06051=1082.787,93.798,-65.194,174.519,21.287,153.556
C06052=1082.781,93.548,-65.176,174.517,21.284,153.556
C06053=1082.776,93.299,-65.158,174.516,21.283,153.556
C06054=1082.769,93.050,-65.139,174.513,21.280,153.556
C06055=1082.764,92.801,-65.122,174.512,21.278,153.556
C06056=1082.758,92.552,-65.104,174.510,21.276,153.555
C06057=1082.753,92.302,-65.086,174.509,21.274,153.555
C06058=1082.748,92.053,-65.068,174.506,21.271,153.555
C06059=1082.741,91.803,-65.050,174.505,21.270,153.555
C06060=1082.736,91.554,-65.032,174.503,21.268,153.555
C06061=1082.731,91.305,-65.014,174.501,21.266,153.555
C06062=1082.725,91.055,-64.996,174.499,21.263,153.555
C06063=1082.719,90.806,-64.978,174.498,21.261,153.554
C06064=1082.713,90.557,-64.960,174.496,21.259,153.554
C06065=1082.708,90.308,-64.943,174.494,21.257,153.554
C06066=1082.702,90.058,-64.925,174.493,21.255,153.554
C06067=1082.696,89.809,-64.907,174.491,21.253,153.554
C06068=1082.690,89.560,-64.889,174.489,21.251,153.554
C06069=1082.684,89.311,-64.871,174.487,21.249,153.554
C06070=1082.678,89.062,-64.854,174.486,21.247,153.554
C06071=1082.672,88.812,-64.836,174.483,21.244,153.553
C06072=1082.667,88.563,-64.818,174.482,21.243,153.553
C06073=1082.661,88.314,-64.800,174.480,21.240,153.553
C06074=1082.655,88.064,-64.783,174.478,21.238,153.553
C06075=1082.650,87.815,-64.765,174.476,21.236,153.553
C06076=1082.644,87.566,-64.747,174.475,21.234,153.553
C06077=1082.639,87.316,-64.729,174.473,21.232,153.553
C06078=1082.633,87.067,-64.711,174.471,21.230,153.552
C06079=1082.627,86.817,-64.693,174.469,21.228,153.552
C06080=1082.622,86.568,-64.676,174.468,21.226,153.552
C06081=1082.616,86.319,-64.658,174.465,21.223,153.552
C06082=1082.610,86.069,-64.640,174.464,21.221,153.552
C06083=1082.604,85.820,-64.623,174.463,21.219,153.552
C06084=1082.599,85.571,-64.605,174.461,21.217,153.551
C06085=1082.593,85.321,-64.587,174.459,21.215,153.551
C06086=1082.588,85.072,-64.570,174.457,21.213,153.551
C06087=1082.582,84.823,-64.553,174.456,21.211,153.551
C06088=1082.576,84.573,-64.535,174.454,21.208,153.551
C06089=1082.570,84.324,-64.517,174.452,21.206,153.551
C06090=1082.564,84.075,-64.500,174.450,21.204,153.551
C06091=1082.559,83.826,-64.483,174.449,21.202,153.550
C06092=1082.553,83.576,-64.465,174.446,21.200,153.550
C06093=1082.547,83.327,-64.447,174.445,21.198,153.550
C06094=1082.541,83.078,-64.430,174.444,21.196,153.550
C06095=1082.536,82.828,-64.413,174.441,21.194,153.550
C06096=1082.530,82.579,-64.395,174.440,21.192,153.550
C06097=1082.525,82.330,-64.377,174.438,21.189,153.550
C06098=1082.519,82.081,-64.360,174.437,21.188,153.549
C06099=1082.513,81.831,-64.342,174.434,21.185,153.549
C06100=1082.508,81.581,-64.325,174.433,21.183,153.549
C06101=1082.502,81.332,-64.307,174.431,21.180,153.549
C06102=1082.497,81.083,-64.290,174.430,21.178,153.549
C06103=1082.491,80.834,-64.272,174.427,21.176,153.548
C06104=1082.485,80.585,-64.254,174.426,21.174,153.548
C06105=1082.480,80.335,-64.238,174.425,21.172,153.548
C06106=1082.474,80.086,-64.220,174.423,21.170,153.548
C06107=1082.468,79.836,-64.202,174.421,21.168,153.548
C06108=1082.462,79.557,-64.183,174.419,21.165,153.548
C06109=1082.456,79.278,-64.164,174.417,21.163,153.548
C06110=1082.449,78.999,-64.144,174.416,21.160,153.547
C06111=1082.443,78.719,-64.125,174.414,21.158,153.547
C06112=1082.437,78.470,-64.107,174.411,21.156,153.547
C06113=1082.432,78.221,-64.090,174.410,21.154,153.547
C06114=1082.426,77.971,-64.073,174.408,21.151,153.547
C06115=1082.420,77.722,-64.056,174.407,21.149,153.546
C06116=1082.414,77.472,-64.038,174.405,21.147,153.546
C06117=1082.409,77.223,-64.021,174.403,21.145,153.546
C06118=1082.403,76.974,-64.004,174.402,21.143,153.546
C06119=1082.397,76.725,-63.986,174.399,21.141,153.546
C06120=1082.391,76.475,-63.969,174.398,21.139,153.546
C06121=1082.386,76.226,-63.952,174.396,21.136,153.546
C06122=1082.380,75.976,-63.935,174.395,21.134,153.545
C06123=1082.374,75.727,-63.918,174.393,21.132,153.545
C06124=1082.369,75.478,-63.900,174.391,21.130,153.545
C06125=1082.362,75.228,-63.884,174.390,21.128,153.545
C06126=1082.357,74.979,-63.866,174.388,21.126,153.545
C06127=1082.352,74.729,-63.849,174.386,21.124,153.545
C06128=1082.346,74.480,-63.832,174.384,21.121,153.544
C06129=1082.340,74.232,-63.815,174.383,21.119,153.544
C06130=1082.334,73.981,-63.797,174.381,21.117,153.544
C06131=1082.328,73.732,-63.780,174.379,21.115,153.544
C06132=1082.322,73.483,-63.764,174.378,21.113,153.544
C06133=1082.317,73.234,-63.746,174.376,21.111,153.544
C06134=1082.312,72.984,-63.729,174.375,21.108,153.543
C06135=1082.305,72.736,-63.712,174.373,21.106,153.543
C06136=1082.300,72.486,-63.695,174.371,21.104,153.543
C06137=1082.294,72.236,-63.677,174.370,21.102,153.543
C06138=1082.288,71.987,-63.661,174.368,21.099,153.543
C06139=1082.283,71.738,-63.644,174.366,21.097,153.543
C06140=1082.277,71.488,-63.627,174.364,21.095,153.542
C06141=1082.271,71.239,-63.610,174.363,21.093,153.542
C06142=1082.266,70.990,-63.593,174.361,21.091,153.542
C06143=1082.261,70.740,-63.576,174.359,21.089,153.542
C06144=1082.255,70.491,-63.559,174.358,21.087,153.542
C06145=1082.249,70.241,-63.542,174.356,21.084,153.541
C06146=1082.242,69.992,-63.525,174.355,21.082,153.541
C06147=1082.237,69.743,-63.508,174.353,21.080,153.541
C06148=1082.232,69.493,-63.491,174.351,21.077,153.541
C06149=1082.226,69.244,-63.474,174.350,21.075,153.541
C06150=1082.221,68.995,-63.457,174.348,21.073,153.541
C06151=1082.214,68.746,-63.440,174.346,21.071,153.540
C06152=1082.209,68.496,-63.424,174.345,21.069,153.540
C06153=1082.203,68.246,-63.407,174.343,21.067,153.540
C06154=1082.197,67.997,-63.389,174.341,21.065,153.540
C06155=1082.191,67.748,-63.373,174.339,21.062,153.540
C06156=1082.186,67.498,-63.356,174.338,21.060,153.540
C06157=1082.180,67.249,-63.339,174.337,21.058,153.539
C06158=1082.174,67.000,-63.322,174.335,21.056,153.539
C06159=1082.168,66.750,-63.306,174.333,21.054,153.539
C06160=1082.163,66.501,-63.289,174.331,21.051,153.539
C06161=1082.157,66.252,-63.272,174.330,21.049,153.539
C06162=1082.152,66.002,-63.256,174.328,21.047,153.539
C06163=1082.146,65.753,-63.239,174.326,21.045,153.538
C06164=1082.140,65.504,-63.222,174.325,21.043,153.538
C06165=1082.134,65.255,-63.205,174.323,21.040,153.538
C06166=1082.128,65.004,-63.189,174.322,21.038,153.538
C06167=1082.123,64.755,-63.172,174.320,21.036,153.538
C06168=1082.116,64.506,-63.155,174.318,21.034,153.538
C06169=1082.111,64.256,-63.138,174.317,21.032,153.537
C06170=1082.105,64.007,-63.122,174.315,21.029,153.537
C06171=1082.099,63.758,-63.106,174.313,21.027,153.537
C06172=1082.093,63.478,-63.087,174.311,21.025,153.537
C06173=1082.086,63.199,-63.068,174.310,21.022,153.537
C06174=1082.079,62.919,-63.050,174.308,21.020,153.536
C06175=1082.073,62.640,-63.031,174.306,21.018,153.536
C06176=1082.067,62.391,-63.015,174.304,21.016,153.536
C06177=1082.061,62.142,-62.998,174.303,21.014,153.536
C06178=1082.055,61.892,-62.981,174.301,21.011,153.536
C06179=1082.049,61.643,-62.965,174.299,21.009,153.536
C06180=1082.044,61.393,-62.948,174.297,21.006,153.535
C06181=1082.038,61.144,-62.932,174.296,21.004,153.535
C06182=1082.032,60.894,-62.915,174.295,21.002,153.535
C06183=1082.026,60.645,-62.899,174.293,21.000,153.535
C06184=1082.020,60.395,-62.883,174.291,20.998,153.535
C06185=1082.015,60.146,-62.866,174.290,20.996,153.535
C06186=1082.009,59.897,-62.849,174.288,20.994,153.534
C06187=1082.003,59.648,-62.833,174.286,20.992,153.534
C06188=1081.997,59.398,-62.816,174.284,20.989,153.534
C06189=1081.991,59.149,-62.800,174.283,20.987,153.534
C06190=1081.985,58.900,-62.784,174.282,20.985,153.534
C06191=1081.980,58.650,-62.767,174.280,20.982,153.533
C06192=1081.974,58.401,-62.751,174.278,20.980,153.533
C06193=1081.968,58.151,-62.734,174.277,20.979,153.533
C06194=1081.962,57.902,-62.718,174.275,20.976,153.533
C06195=1081.956,57.653,-62.702,174.274,20.974,153.533
C06196=1081.951,57.403,-62.685,174.271,20.972,153.533
C06197=1081.945,57.154,-62.669,174.270,20.970,153.533
C06198=1081.939,56.904,-62.653,174.269,20.967,153.532
C06199=1081.933,56.655,-62.636,174.267,20.965,153.532
C06200=1081.927,56.406,-62.620,174.265,20.963,153.532
C06201=1081.922,56.156,-62.603,174.264,20.961,153.532
C06202=1081.916,55.907,-62.587,174.262,20.959,153.532
C06203=1081.910,55.657,-62.571,174.261,20.957,153.531
C06204=1081.904,55.408,-62.554,174.259,20.954,153.531
C06205=1081.899,55.159,-62.539,174.257,20.952,153.531
C06206=1081.893,54.909,-62.523,174.256,20.950,153.531
C06207=1081.888,54.660,-62.506,174.254,20.947,153.531
C06208=1081.882,54.410,-62.490,174.252,20.945,153.531
C06209=1081.876,54.161,-62.474,174.251,20.943,153.530
C06210=1081.870,53.912,-62.457,174.249,20.940,153.530
C06211=1081.864,53.662,-62.441,174.248,20.938,153.530
C06212=1081.858,53.413,-62.425,174.247,20.937,153.530
C06213=1081.852,53.164,-62.409,174.244,20.934,153.530
C06214=1081.847,52.913,-62.393,174.243,20.932,153.529
C06215=1081.841,52.664,-62.376,174.241,20.929,153.529
C06216=1081.836,52.415,-62.360,174.240,20.927,153.529
C06217=1081.830,52.166,-62.344,174.238,20.925,153.529
C06218=1081.824,51.917,-62.328,174.236,20.923,153.529
C06219=1081.818,51.667,-62.312,174.235,20.920,153.528
C06220=1081.812,51.417,-62.296,174.234,20.918,153.528
C06221=1081.807,51.168,-62.280,174.232,20.916,153.528
C06222=1081.801,50.918,-62.263,174.230,20.914,153.528
C06223=1081.796,50.670,-62.247,174.229,20.912,153.528
C06224=1081.790,50.420,-62.232,174.227,20.909,153.527
C06225=1081.784,50.170,-62.215,174.226,20.907,153.527
C06226=1081.778,49.921,-62.199,174.224,20.905,153.527
C06227=1081.772,49.672,-62.183,174.222,20.903,153.527
C06228=1081.767,49.422,-62.167,174.221,20.900,153.527
C06229=1081.761,49.173,-62.151,174.220,20.898,153.526
C06230=1081.756,48.924,-62.135,174.218,20.896,153.526
C06231=1081.750,48.674,-62.119,174.217,20.893,153.526
C06232=1081.744,48.424,-62.103,174.214,20.891,153.526
C06233=1081.739,48.175,-62.086,174.213,20.889,153.526
C06234=1081.733,47.926,-62.071,174.212,20.887,153.526
C06235=1081.728,47.676,-62.055,174.210,20.884,153.525
C06236=1081.721,47.396,-62.036,174.208,20.882,153.525
C06237=1081.714,47.117,-62.019,174.207,20.879,153.525
C06238=1081.708,46.838,-62.002,174.205,20.877,153.525
C06239=1081.702,46.557,-61.983,174.203,20.874,153.524
C06240=1081.696,46.308,-61.967,174.202,20.872,153.524
C06241=1081.691,46.059,-61.951,174.200,20.870,153.524
C06242=1081.685,45.809,-61.936,174.199,20.867,153.524
C06243=1081.679,45.560,-61.919,174.197,20.865,153.524
C06244=1081.673,45.310,-61.903,174.195,20.863,153.523
C06245=1081.668,45.061,-61.888,174.194,20.860,153.523
C06246=1081.662,44.812,-61.872,174.193,20.859,153.523
C06247=1081.657,44.562,-61.856,174.191,20.856,153.523
C06248=1081.651,44.312,-61.840,174.189,20.854,153.523
C06249=1081.646,44.063,-61.825,174.188,20.852,153.522
C06250=1081.640,43.814,-61.808,174.186,20.849,153.522
C06251=1081.634,43.565,-61.792,174.185,20.847,153.522
C06252=1081.628,43.315,-61.777,174.184,20.845,153.522
C06253=1081.623,43.066,-61.761,174.181,20.842,153.522
C06254=1081.616,42.816,-61.746,174.180,20.840,153.521
C06255=1081.610,42.567,-61.730,174.179,20.838,153.521
C06256=1081.605,42.317,-61.714,174.177,20.835,153.521
C06257=1081.599,42.068,-61.698,174.176,20.833,153.521
C06258=1081.594,41.818,-61.683,174.174,20.832,153.521
C06259=1081.588,41.569,-61.666,174.172,20.829,153.521
C06260=1081.582,41.319,-61.651,174.171,20.827,153.520
C06261=1081.576,41.071,-61.636,174.170,20.825,153.520
C06262=1081.570,40.821,-61.620,174.167,20.822,153.520
C06263=1081.565,40.571,-61.604,174.166,20.820,153.520
C06264=1081.559,40.322,-61.589,174.165,20.818,153.519
C06265=1081.554,40.072,-61.573,174.163,20.815,153.519
C06266=1081.547,39.823,-61.557,174.162,20.813,153.519
C06267=1081.541,39.573,-61.542,174.160,20.811,153.519
C06268=1081.536,39.324,-61.526,174.158,20.808,153.519
C06269=1081.530,39.074,-61.510,174.157,20.806,153.519
C06270=1081.525,38.825,-61.495,174.156,20.804,153.518
C06271=1081.519,38.576,-61.479,174.154,20.802,153.518
C06272=1081.513,38.326,-61.464,174.152,20.800,153.518
C06273=1081.507,38.076,-61.448,174.151,20.798,153.518
C06274=1081.502,37.828,-61.433,174.149,20.795,153.517
C06275=1081.496,37.578,-61.418,174.148,20.793,153.517
C06276=1081.490,37.329,-61.401,174.147,20.791,153.517
C06277=1081.484,37.079,-61.386,174.144,20.788,153.517
C06278=1081.478,36.830,-61.371,174.143,20.786,153.517
C06279=1081.472,36.580,-61.355,174.142,20.784,153.516
C06280=1081.467,36.330,-61.339,174.141,20.782,153.516
C06281=1081.461,36.081,-61.325,174.138,20.779,153.516
C06282=1081.455,35.831,-61.309,174.137,20.777,153.516
C06283=1081.449,35.582,-61.293,174.136,20.775,153.516
C06284=1081.443,35.332,-61.278,174.134,20.773,153.516
C06285=1081.438,35.083,-61.263,174.133,20.771,153.515
C06286=1081.432,34.834,-61.247,174.131,20.769,153.515
C06287=1081.426,34.584,-61.232,174.129,20.766,153.515
C06288=1081.421,34.335,-61.217,174.128,20.764,153.515
C06289=1081.414,34.085,-61.202,174.127,20.762,153.515
C06290=1081.408,33.836,-61.185,174.125,20.759,153.514
C06291=1081.403,33.587,-61.170,174.123,20.757,153.514
C06292=1081.397,33.337,-61.155,174.122,20.755,153.514
C06293=1081.391,33.087,-61.140,174.121,20.753,153.514
C06294=1081.385,32.838,-61.125,174.119,20.750,153.514
C06295=1081.379,32.589,-61.109,174.118,20.748,153.513
C06296=1081.374,32.339,-61.094,174.116,20.746,153.513
C06297=1081.368,32.090,-61.079,174.114,20.743,153.513
C06298=1081.362,31.840,-61.063,174.113,20.741,153.513
C06299=1081.357,31.591,-61.049,174.112,20.739,153.513
C06300=1081.350,31.311,-61.031,174.110,20.737,153.512
C06301=1081.344,31.031,-61.013,174.108,20.734,153.512
C06302=1081.337,30.752,-60.997,174.106,20.732,153.512
C06303=1081.331,30.472,-60.980,174.104,20.729,153.512
C06304=1081.325,30.223,-60.964,174.103,20.727,153.512
C06305=1081.319,29.974,-60.949,174.102,20.724,153.511
C06306=1081.313,29.724,-60.934,174.101,20.722,153.511
C06307=1081.308,29.475,-60.919,174.098,20.720,153.511
C06308=1081.302,29.225,-60.903,174.097,20.717,153.511
C06309=1081.296,28.976,-60.889,174.096,20.715,153.510
C06310=1081.290,28.726,-60.873,174.094,20.713,153.510
C06311=1081.285,28.477,-60.859,174.093,20.711,153.510
C06312=1081.279,28.227,-60.843,174.091,20.708,153.510
C06313=1081.273,27.977,-60.828,174.089,20.706,153.510
C06314=1081.268,27.728,-60.813,174.088,20.704,153.510
C06315=1081.261,27.478,-60.798,174.087,20.702,153.509
C06316=1081.255,27.229,-60.784,174.086,20.700,153.509
C06317=1081.250,26.979,-60.768,174.083,20.697,153.509
C06318=1081.243,26.730,-60.753,174.082,20.695,153.509
C06319=1081.238,26.481,-60.738,174.081,20.693,153.509
C06320=1081.232,26.231,-60.723,174.079,20.690,153.508
C06321=1081.226,25.982,-60.708,174.078,20.688,153.508
C06322=1081.221,25.732,-60.693,174.076,20.686,153.508
C06323=1081.215,25.483,-60.678,174.075,20.684,153.508
C06324=1081.209,25.233,-60.663,174.073,20.681,153.508
C06325=1081.203,24.983,-60.648,174.072,20.679,153.507
C06326=1081.197,24.734,-60.633,174.070,20.677,153.507
C06327=1081.191,24.484,-60.618,174.068,20.675,153.507
C06328=1081.186,24.235,-60.603,174.067,20.672,153.507
C06329=1081.179,23.986,-60.588,174.066,20.670,153.507
C06330=1081.174,23.737,-60.573,174.065,20.668,153.506
C06331=1081.168,23.487,-60.558,174.062,20.666,153.506
C06332=1081.162,23.238,-60.543,174.061,20.664,153.506
C06333=1081.156,22.988,-60.528,174.060,20.662,153.506
C06334=1081.151,22.739,-60.513,174.059,20.660,153.506
C06335=1081.144,22.489,-60.499,174.057,20.657,153.506
C06336=1081.139,22.239,-60.484,174.055,20.655,153.505
C06337=1081.133,21.990,-60.469,174.054,20.653,153.505
C06338=1081.127,21.741,-60.454,174.052,20.650,153.505
C06339=1081.122,21.491,-60.439,174.051,20.648,153.505
C06340=1081.116,21.242,-60.424,174.050,20.646,153.504
C06341=1081.109,20.992,-60.409,174.048,20.644,153.504
C06342=1081.105,20.742,-60.395,174.046,20.641,153.504
C06343=1081.098,20.493,-60.380,174.045,20.639,153.504
C06344=1081.093,20.244,-60.365,174.044,20.637,153.504
C06345=1081.087,19.994,-60.350,174.042,20.634,153.504
C06346=1081.081,19.745,-60.335,174.041,20.632,153.503
C06347=1081.075,19.495,-60.321,174.039,20.630,153.503
C06348=1081.069,19.246,-60.306,174.038,20.628,153.503
C06349=1081.063,18.996,-60.291,174.036,20.625,153.503
C06350=1081.058,18.747,-60.276,174.035,20.623,153.502
C06351=1081.052,18.496,-60.262,174.033,20.621,153.502
C06352=1081.046,18.247,-60.247,174.032,20.619,153.502
C06353=1081.040,17.998,-60.233,174.030,20.617,153.502
C06354=1081.035,17.749,-60.217,174.029,20.614,153.502
C06355=1081.029,17.499,-60.204,174.028,20.612,153.501
C06356=1081.023,17.249,-60.189,174.026,20.610,153.501
C06357=1081.017,17.000,-60.174,174.024,20.608,153.501
C06358=1081.011,16.751,-60.159,174.023,20.605,153.501
C06359=1081.005,16.501,-60.145,174.022,20.603,153.501
C06360=1080.999,16.251,-60.130,174.020,20.601,153.501
C06361=1080.994,16.002,-60.115,174.018,20.599,153.500
C06362=1080.988,15.753,-60.101,174.017,20.596,153.500
C06363=1080.982,15.503,-60.086,174.016,20.594,153.500
C06364=1080.975,15.225,-60.070,174.014,20.592,153.500
C06365=1080.969,14.946,-60.053,174.013,20.589,153.499
C06366=1080.963,14.669,-60.038,174.011,20.587,153.499
C06367=1080.956,14.390,-60.021,174.009,20.584,153.499
C06368=1080.950,14.141,-60.007,174.007,20.582,153.499
C06369=1080.944,13.891,-59.993,174.006,20.580,153.499
C06370=1080.938,13.641,-59.978,174.005,20.577,153.498
C06371=1080.932,13.392,-59.963,174.004,20.575,153.498
C06372=1080.927,13.143,-59.949,174.001,20.573,153.498
C06373=1080.920,12.893,-59.934,174.000,20.571,153.498
C06374=1080.915,12.644,-59.920,173.999,20.569,153.498
C06375=1080.909,12.394,-59.906,173.998,20.567,153.497
C06376=1080.903,12.144,-59.892,173.996,20.564,153.497
C06377=1080.897,11.895,-59.877,173.994,20.562,153.497
C06378=1080.891,11.646,-59.862,173.993,20.560,153.497
C06379=1080.885,11.396,-59.848,173.992,20.558,153.497
C06380=1080.879,11.147,-59.833,173.990,20.556,153.497
C06381=1080.874,10.897,-59.819,173.988,20.553,153.496
C06382=1080.867,10.647,-59.804,173.987,20.551,153.496
C06383=1080.862,10.398,-59.791,173.986,20.549,153.496
C06384=1080.856,10.149,-59.776,173.984,20.547,153.496
C06385=1080.850,9.899,-59.762,173.982,20.545,153.496
C06386=1080.844,9.650,-59.747,173.981,20.542,153.495
C06387=1080.838,9.399,-59.733,173.980,20.540,153.495
C06388=1080.831,9.151,-59.719,173.978,20.538,153.495
C06389=1080.826,8.901,-59.705,173.977,20.536,153.495
C06390=1080.820,8.651,-59.690,173.976,20.533,153.495
C06391=1080.814,8.402,-59.676,173.974,20.531,153.495
C06392=1080.809,8.152,-59.662,173.972,20.529,153.494
C06393=1080.802,7.903,-59.648,173.971,20.527,153.494
C06394=1080.797,7.653,-59.634,173.970,20.525,153.494
C06395=1080.791,7.404,-59.619,173.968,20.522,153.494
C06396=1080.785,7.154,-59.605,173.966,20.520,153.494
C06397=1080.779,6.905,-59.590,173.965,20.518,153.493
C06398=1080.774,6.655,-59.576,173.964,20.516,153.493
C06399=1080.768,6.405,-59.562,173.962,20.514,153.493
C06400=1080.762,6.156,-59.548,173.960,20.511,153.493
C06401=1080.756,5.907,-59.534,173.959,20.509,153.493
C06402=1080.750,5.656,-59.520,173.958,20.507,153.492
C06403=1080.744,5.408,-59.506,173.957,20.505,153.492
C06404=1080.738,5.158,-59.492,173.956,20.503,153.492
C06405=1080.733,4.908,-59.478,173.953,20.500,153.492
C06406=1080.726,4.659,-59.463,173.952,20.498,153.492
C06407=1080.721,4.409,-59.449,173.951,20.496,153.492
C06408=1080.715,4.160,-59.435,173.949,20.494,153.491
C06409=1080.709,3.910,-59.420,173.948,20.491,153.491
C06410=1080.703,3.661,-59.407,173.946,20.489,153.491
C06411=1080.697,3.411,-59.393,173.945,20.487,153.491
C06412=1080.692,3.162,-59.378,173.944,20.485,153.491
C06413=1080.685,2.912,-59.364,173.942,20.482,153.490
C06414=1080.680,2.662,-59.350,173.940,20.480,153.490
C06415=1080.675,2.413,-59.337,173.939,20.478,153.490
C06416=1080.669,2.164,-59.322,173.938,20.476,153.490
C06417=1080.662,1.914,-59.308,173.936,20.473,153.490
C06418=1080.656,1.664,-59.294,173.935,20.471,153.489
C06419=1080.651,1.415,-59.281,173.933,20.469,153.489
C06420=1080.645,1.166,-59.266,173.932,20.467,153.489
C06421=1080.639,0.915,-59.252,173.931,20.465,153.489
C06422=1080.634,0.666,-59.238,173.929,20.462,153.489
C06423=1080.628,0.416,-59.224,173.928,20.460,153.488
C06424=1080.622,0.167,-59.211,173.926,20.458,153.488
C06425=1080.616,-0.082,-59.196,173.925,20.456,153.488
C06426=1080.610,-0.332,-59.182,173.923,20.454,153.488
C06427=1080.605,-0.582,-59.168,173.922,20.452,153.488
C06428=1080.598,-0.858,-59.153,173.920,20.450,153.487
C06429=1080.592,-1.134,-59.138,173.919,20.447,153.487
C06430=1080.586,-1.410,-59.122,173.917,20.445,153.487
C06431=1080.579,-1.686,-59.107,173.915,20.442,153.487
C06432=1080.573,-1.936,-59.093,173.914,20.440,153.487
C06433=1080.568,-2.185,-59.079,173.913,20.438,153.486
C06434=1080.562,-2.435,-59.065,173.912,20.435,153.486
C06435=1080.556,-2.685,-59.051,173.910,20.433,153.486
C06436=1080.550,-2.934,-59.038,173.908,20.431,153.486
C06437=1080.545,-3.184,-59.024,173.907,20.429,153.486
C06438=1080.539,-3.433,-59.010,173.906,20.427,153.485
C06439=1080.534,-3.683,-58.996,173.905,20.424,153.485
C06440=1080.526,-3.932,-58.982,173.902,20.422,153.485
C06441=1080.521,-4.182,-58.968,173.901,20.420,153.485
C06442=1080.515,-4.431,-58.955,173.900,20.418,153.485
C06443=1080.509,-4.681,-58.941,173.899,20.416,153.485
C06444=1080.503,-4.930,-58.927,173.896,20.413,153.484
C06445=1080.497,-5.180,-58.913,173.895,20.411,153.484
C06446=1080.492,-5.430,-58.899,173.894,20.409,153.484
C06447=1080.485,-5.679,-58.886,173.893,20.407,153.484
C06448=1080.480,-5.929,-58.872,173.891,20.405,153.484
C06449=1080.474,-6.178,-58.859,173.889,20.402,153.483
C06450=1080.468,-6.428,-58.845,173.888,20.400,153.483
C06451=1080.461,-6.678,-58.831,173.887,20.398,153.483
C06452=1080.456,-6.927,-58.818,173.885,20.396,153.483
C06453=1080.450,-7.176,-58.804,173.884,20.394,153.483
C06454=1080.444,-7.426,-58.790,173.882,20.392,153.483
C06455=1080.438,-7.675,-58.777,173.881,20.389,153.482
C06456=1080.432,-7.926,-58.763,173.880,20.387,153.482
C06457=1080.426,-8.175,-58.749,173.878,20.385,153.482
C06458=1080.420,-8.424,-58.736,173.876,20.383,153.482
C06459=1080.415,-8.675,-58.723,173.875,20.381,153.482
C06460=1080.409,-8.924,-58.709,173.874,20.379,153.482
C06461=1080.403,-9.173,-58.695,173.872,20.377,153.481
C06462=1080.397,-9.423,-58.682,173.871,20.375,153.481
C06463=1080.392,-9.672,-58.668,173.869,20.373,153.481
C06464=1080.385,-9.922,-58.655,173.868,20.370,153.481
C06465=1080.379,-10.172,-58.641,173.867,20.368,153.481
C06466=1080.373,-10.421,-58.628,173.865,20.366,153.480
C06467=1080.368,-10.671,-58.614,173.864,20.364,153.480
C06468=1080.361,-10.920,-58.600,173.862,20.362,153.480
C06469=1080.356,-11.170,-58.587,173.861,20.360,153.480
C06470=1080.350,-11.419,-58.574,173.859,20.358,153.480
C06471=1080.345,-11.669,-58.560,173.858,20.356,153.480
C06472=1080.338,-11.918,-58.547,173.857,20.353,153.479
C06473=1080.333,-12.168,-58.533,173.855,20.351,153.479
C06474=1080.327,-12.417,-58.520,173.854,20.349,153.479
C06475=1080.321,-12.667,-58.507,173.852,20.347,153.479
C06476=1080.315,-12.917,-58.493,173.851,20.345,153.479
C06477=1080.309,-13.167,-58.479,173.850,20.343,153.479
C06478=1080.303,-13.416,-58.466,173.848,20.340,153.478
C06479=1080.297,-13.665,-58.453,173.846,20.338,153.478
C06480=1080.292,-13.915,-58.439,173.845,20.336,153.478
C06481=1080.285,-14.165,-58.426,173.844,20.334,153.478
C06482=1080.280,-14.414,-58.412,173.843,20.332,153.478
C06483=1080.274,-14.664,-58.399,173.841,20.329,153.477
C06484=1080.269,-14.914,-58.386,173.839,20.327,153.477
C06485=1080.262,-15.163,-58.373,173.838,20.325,153.477
C06486=1080.256,-15.412,-58.359,173.837,20.323,153.477
C06487=1080.251,-15.662,-58.345,173.835,20.321,153.477
C06488=1080.245,-15.912,-58.333,173.833,20.319,153.477
C06489=1080.238,-16.161,-58.320,173.832,20.317,153.476
C06490=1080.233,-16.411,-58.306,173.831,20.315,153.476
C06491=1080.227,-16.660,-58.293,173.829,20.313,153.476
C06492=1080.220,-16.935,-58.279,173.827,20.310,153.476
C06493=1080.213,-17.210,-58.263,173.826,20.308,153.476
C06494=1080.207,-17.484,-58.249,173.825,20.306,153.476
C06495=1080.201,-17.759,-58.235,173.823,20.303,153.475
C06496=1080.195,-18.009,-58.222,173.821,20.301,153.475
C06497=1080.188,-18.258,-58.209,173.820,20.299,153.475
C06498=1080.183,-18.507,-58.195,173.819,20.297,153.475
C06499=1080.177,-18.757,-58.182,173.818,20.295,153.475
C06500=1080.171,-19.007,-58.169,173.816,20.293,153.475
C06501=1080.165,-19.256,-58.156,173.814,20.291,153.474
C06502=1080.159,-19.506,-58.143,173.813,20.289,153.474
C06503=1080.153,-19.755,-58.129,173.812,20.287,153.474
C06504=1080.147,-20.005,-58.117,173.810,20.285,153.474
C06505=1080.141,-20.254,-58.104,173.808,20.283,153.474
C06506=1080.136,-20.504,-58.090,173.807,20.281,153.474
C06507=1080.130,-20.754,-58.077,173.806,20.279,153.473
C06508=1080.124,-21.003,-58.064,173.804,20.277,153.473
C06509=1080.118,-21.253,-58.051,173.803,20.275,153.473
C06510=1080.112,-21.503,-58.037,173.802,20.273,153.473
C06511=1080.106,-21.752,-58.025,173.800,20.270,153.473
C06512=1080.100,-22.002,-58.012,173.799,20.268,153.473
C06513=1080.094,-22.252,-57.999,173.797,20.266,153.472
C06514=1080.088,-22.501,-57.986,173.796,20.264,153.472
C06515=1080.083,-22.751,-57.973,173.795,20.262,153.472
C06516=1080.077,-23.000,-57.959,173.793,20.259,153.472
C06517=1080.070,-23.250,-57.946,173.791,20.257,153.472
C06518=1080.064,-23.499,-57.934,173.790,20.255,153.472
C06519=1080.059,-23.749,-57.921,173.789,20.253,153.471
C06520=1080.053,-23.999,-57.907,173.788,20.251,153.471
C06521=1080.048,-24.248,-57.895,173.786,20.249,153.471
C06522=1080.042,-24.497,-57.882,173.784,20.247,153.471
C06523=1080.036,-24.747,-57.869,173.783,20.245,153.471
C06524=1080.029,-24.997,-57.856,173.782,20.243,153.471
C06525=1080.023,-25.246,-57.843,173.780,20.241,153.470
C06526=1080.018,-25.496,-57.829,173.779,20.239,153.470
C06527=1080.012,-25.746,-57.817,173.778,20.237,153.470
C06528=1080.006,-25.996,-57.804,173.776,20.234,153.470
C06529=1080.000,-26.245,-57.791,173.774,20.232,153.470
C06530=1079.994,-26.495,-57.779,173.773,20.230,153.470
C06531=1079.988,-26.743,-57.766,173.772,20.228,153.469
C06532=1079.983,-26.994,-57.753,173.770,20.226,153.469
C06533=1079.977,-27.244,-57.740,173.769,20.225,153.469
C06534=1079.971,-27.493,-57.727,173.767,20.222,153.469
C06535=1079.965,-27.743,-57.714,173.766,20.220,153.469
C06536=1079.959,-27.992,-57.701,173.764,20.218,153.469
C06537=1079.953,-28.242,-57.688,173.763,20.216,153.469
C06538=1079.947,-28.492,-57.676,173.762,20.214,153.468
C06539=1079.940,-28.741,-57.663,173.760,20.212,153.468
C06540=1079.934,-28.991,-57.651,173.758,20.210,153.468
C06541=1079.928,-29.240,-57.638,173.757,20.208,153.468
C06542=1079.922,-29.490,-57.625,173.756,20.206,153.468
C06543=1079.917,-29.739,-57.613,173.754,20.204,153.468
C06544=1079.911,-29.989,-57.600,173.753,20.202,153.468
C06545=1079.905,-30.238,-57.587,173.752,20.200,153.467
C06546=1079.899,-30.488,-57.574,173.750,20.198,153.467
C06547=1079.893,-30.738,-57.562,173.748,20.196,153.467
C06548=1079.887,-30.988,-57.549,173.747,20.194,153.467
C06549=1079.881,-31.237,-57.536,173.746,20.192,153.467
C06550=1079.875,-31.487,-57.523,173.744,20.190,153.467
C06551=1079.870,-31.736,-57.511,173.743,20.188,153.467
C06552=1079.864,-31.986,-57.498,173.742,20.186,153.466
C06553=1079.858,-32.235,-57.485,173.740,20.184,153.466
C06554=1079.852,-32.485,-57.473,173.738,20.182,153.466
C06555=1079.846,-32.735,-57.460,173.737,20.180,153.466
C06556=1079.839,-33.009,-57.446,173.736,20.178,153.466
C06557=1079.833,-33.282,-57.433,173.734,20.175,153.466
C06558=1079.826,-33.556,-57.419,173.732,20.173,153.466
C06559=1079.819,-33.829,-57.405,173.731,20.171,153.465
C06560=1079.813,-34.079,-57.392,173.729,20.169,153.465
C06561=1079.808,-34.329,-57.380,173.728,20.167,153.465
C06562=1079.802,-34.579,-57.367,173.726,20.165,153.465
C06563=1079.796,-34.828,-57.355,173.725,20.163,153.465
C06564=1079.790,-35.078,-57.342,173.724,20.162,153.465
C06565=1079.785,-35.328,-57.330,173.722,20.160,153.465
C06566=1079.778,-35.577,-57.316,173.721,20.158,153.464
C06567=1079.772,-35.827,-57.305,173.719,20.155,153.464
C06568=1079.766,-36.076,-57.292,173.718,20.153,153.464
C06569=1079.760,-36.326,-57.280,173.716,20.151,153.464
C06570=1079.755,-36.576,-57.267,173.715,20.149,153.464
C06571=1079.749,-36.826,-57.255,173.714,20.148,153.464
C06572=1079.743,-37.075,-57.243,173.712,20.146,153.464
C06573=1079.737,-37.325,-57.230,173.711,20.144,153.463
C06574=1079.731,-37.574,-57.217,173.709,20.141,153.463
C06575=1079.725,-37.824,-57.204,173.708,20.139,153.463
C06576=1079.719,-38.073,-57.193,173.706,20.137,153.463
C06577=1079.713,-38.323,-57.180,173.705,20.136,153.463
C06578=1079.707,-38.572,-57.167,173.704,20.134,153.463
C06579=1079.702,-38.822,-57.155,173.702,20.132,153.463
C06580=1079.696,-39.071,-57.143,173.701,20.130,153.462
C06581=1079.690,-39.321,-57.131,173.700,20.128,153.462
C06582=1079.684,-39.571,-57.118,173.697,20.126,153.462
C06583=1079.678,-39.821,-57.106,173.696,20.124,153.462
C06584=1079.671,-40.070,-57.094,173.695,20.122,153.462
C06585=1079.666,-40.320,-57.081,173.694,20.120,153.462
C06586=1079.660,-40.569,-57.069,173.692,20.118,153.462
C06587=1079.654,-40.819,-57.056,173.691,20.116,153.462
C06588=1079.647,-41.069,-57.044,173.690,20.114,153.461
C06589=1079.642,-41.318,-57.032,173.687,20.112,153.461
C06590=1079.636,-41.568,-57.020,173.686,20.110,153.461
C06591=1079.629,-41.818,-57.008,173.685,20.108,153.461
C06592=1079.624,-42.067,-56.995,173.683,20.106,153.461
C06593=1079.618,-42.317,-56.983,173.682,20.105,153.461
C06594=1079.612,-42.566,-56.971,173.681,20.103,153.461
C06595=1079.606,-42.816,-56.958,173.679,20.101,153.461
C06596=1079.600,-43.066,-56.946,173.678,20.099,153.461
C06597=1079.594,-43.315,-56.935,173.676,20.097,153.460
C06598=1079.588,-43.565,-56.922,173.674,20.095,153.460
C06599=1079.582,-43.815,-56.910,173.673,20.093,153.460
C06600=1079.576,-44.064,-56.898,173.672,20.091,153.460
C06601=1079.570,-44.314,-56.886,173.670,20.089,153.460
C06602=1079.564,-44.564,-56.873,173.669,20.087,153.460
C06603=1079.558,-44.813,-56.861,173.668,20.086,153.460
C06604=1079.552,-45.063,-56.849,173.666,20.084,153.460
C06605=1079.546,-45.312,-56.837,173.665,20.082,153.459
C06606=1079.540,-45.563,-56.825,173.663,20.080,153.459
C06607=1079.535,-45.812,-56.813,173.661,20.078,153.459
C06608=1079.528,-46.061,-56.801,173.660,20.076,153.459
C06609=1079.522,-46.311,-56.789,173.659,20.074,153.459
C06610=1079.517,-46.561,-56.776,173.657,20.072,153.459
C06611=1079.510,-46.810,-56.764,173.656,20.070,153.459
C06612=1079.505,-47.061,-56.753,173.655,20.068,153.458
C06613=1079.499,-47.309,-56.741,173.653,20.067,153.458
C06614=1079.493,-47.559,-56.728,173.651,20.064,153.458
C06615=1079.487,-47.809,-56.716,173.650,20.062,153.458
C06616=1079.481,-48.058,-56.704,173.649,20.061,153.458
C06617=1079.475,-48.309,-56.692,173.647,20.059,153.458
C06618=1079.469,-48.557,-56.681,173.646,20.057,153.458
C06619=1079.463,-48.807,-56.668,173.644,20.055,153.458
C06620=1079.457,-49.082,-56.655,173.643,20.053,153.458
C06621=1079.450,-49.356,-56.642,173.641,20.051,153.458
C06622=1079.444,-49.630,-56.629,173.640,20.049,153.457
C06623=1079.437,-49.904,-56.616,173.639,20.047,153.457
C06624=1079.432,-50.154,-56.604,173.637,20.045,153.457
C06625=1079.426,-50.404,-56.591,173.635,20.043,153.457
C06626=1079.420,-50.653,-56.580,173.633,20.042,153.457
C06627=1079.413,-50.903,-56.568,173.632,20.040,153.457
C06628=1079.407,-51.153,-56.556,173.631,20.038,153.457
C06629=1079.401,-51.402,-56.544,173.629,20.036,153.457
C06630=1079.395,-51.652,-56.533,173.628,20.035,153.457
C06631=1079.389,-51.902,-56.521,173.627,20.033,153.456
C06632=1079.383,-52.150,-56.509,173.625,20.031,153.456
C06633=1079.377,-52.401,-56.498,173.624,20.029,153.456
C06634=1079.371,-52.651,-56.485,173.622,20.028,153.456
C06635=1079.365,-52.899,-56.474,173.621,20.026,153.456
C06636=1079.358,-53.150,-56.462,173.619,20.024,153.456
C06637=1079.352,-53.399,-56.450,173.617,20.022,153.456
C06638=1079.346,-53.648,-56.438,173.616,20.020,153.456
C06639=1079.340,-53.899,-56.427,173.615,20.018,153.456
C06640=1079.334,-54.148,-56.414,173.613,20.017,153.456
C06641=1079.328,-54.397,-56.403,173.612,20.015,153.456
C06642=1079.322,-54.647,-56.392,173.610,20.013,153.455
C06643=1079.316,-54.896,-56.380,173.609,20.011,153.455
C06644=1079.310,-55.147,-56.368,173.608,20.010,153.455
C06645=1079.303,-55.396,-56.356,173.606,20.008,153.455
C06646=1079.297,-55.645,-56.345,173.605,20.006,153.455
C06647=1079.292,-55.896,-56.333,173.603,20.004,153.455
C06648=1079.286,-56.145,-56.321,173.601,20.002,153.455
C06649=1079.279,-56.395,-56.310,173.600,20.001,153.455
C06650=1079.273,-56.644,-56.298,173.599,19.999,153.455
C06651=1079.268,-56.894,-56.286,173.597,19.997,153.455
C06652=1079.261,-57.144,-56.274,173.596,19.995,153.455
C06653=1079.255,-57.393,-56.264,173.594,19.994,153.455
C06654=1079.250,-57.643,-56.251,173.593,19.992,153.454
C06655=1079.243,-57.893,-56.240,173.592,19.990,153.454
C06656=1079.237,-58.142,-56.228,173.590,19.988,153.454
C06657=1079.231,-58.392,-56.217,173.589,19.987,153.454
C06658=1079.225,-58.642,-56.205,173.587,19.985,153.454
C06659=1079.219,-58.892,-56.194,173.586,19.983,153.454
C06660=1079.213,-59.141,-56.182,173.584,19.981,153.454
C06661=1079.207,-59.391,-56.171,173.582,19.979,153.454
C06662=1079.201,-59.640,-56.158,173.581,19.978,153.454
C06663=1079.195,-59.890,-56.147,173.580,19.976,153.454
C06664=1079.189,-60.139,-56.136,173.578,19.974,153.454
C06665=1079.183,-60.389,-56.124,173.577,19.973,153.454
C06666=1079.177,-60.639,-56.112,173.575,19.971,153.453
C06667=1079.171,-60.889,-56.101,173.574,19.970,153.453
C06668=1079.165,-61.139,-56.090,173.573,19.968,153.453
C06669=1079.159,-61.388,-56.078,173.571,19.966,153.453
C06670=1079.152,-61.638,-56.067,173.570,19.965,153.453
C06671=1079.147,-61.887,-56.055,173.568,19.963,153.453
C06672=1079.141,-62.137,-56.043,173.567,19.961,153.453
C06673=1079.135,-62.387,-56.033,173.566,19.959,153.453
C06674=1079.128,-62.636,-56.021,173.563,19.957,153.453
C06675=1079.123,-62.886,-56.009,173.562,19.956,153.453
C06676=1079.117,-63.136,-55.998,173.561,19.954,153.453
C06677=1079.111,-63.385,-55.986,173.559,19.952,153.453
C06678=1079.105,-63.635,-55.975,173.558,19.951,153.453
C06679=1079.099,-63.884,-55.963,173.556,19.949,153.452
C06680=1079.094,-64.134,-55.952,173.555,19.947,153.452
C06681=1079.087,-64.384,-55.941,173.553,19.946,153.452
C06682=1079.081,-64.633,-55.929,173.552,19.944,153.452
C06683=1079.075,-64.883,-55.918,173.551,19.942,153.452
C06684=1079.069,-65.159,-55.905,173.549,19.940,153.452
C06685=1079.062,-65.434,-55.893,173.547,19.938,153.452
C06686=1079.056,-65.710,-55.881,173.546,19.936,153.452
C06687=1079.049,-65.985,-55.869,173.544,19.935,153.452
C06688=1079.043,-66.234,-55.857,173.543,19.933,153.452
C06689=1079.037,-66.485,-55.845,173.541,19.931,153.452
C06690=1079.031,-66.734,-55.834,173.540,19.930,153.452
C06691=1079.025,-66.984,-55.822,173.538,19.928,153.452
C06692=1079.019,-67.233,-55.811,173.537,19.926,153.451
C06693=1079.013,-67.483,-55.800,173.536,19.925,153.451
C06694=1079.007,-67.733,-55.789,173.534,19.923,153.451
C06695=1079.002,-67.983,-55.778,173.532,19.921,153.451
C06696=1078.995,-68.232,-55.766,173.531,19.919,153.451
C06697=1078.989,-68.482,-55.755,173.529,19.918,153.451
C06698=1078.984,-68.731,-55.744,173.528,19.916,153.451
C06699=1078.977,-68.981,-55.733,173.526,19.914,153.451
C06700=1078.972,-69.231,-55.722,173.525,19.913,153.451
C06701=1078.965,-69.480,-55.710,173.524,19.911,153.451
C06702=1078.960,-69.730,-55.699,173.522,19.909,153.451
C06703=1078.954,-69.980,-55.688,173.521,19.908,153.451
C06704=1078.948,-70.230,-55.676,173.519,19.906,153.451
C06705=1078.942,-70.479,-55.666,173.518,19.904,153.451
C06706=1078.936,-70.729,-55.655,173.516,19.903,153.451
C06707=1078.930,-70.978,-55.643,173.515,19.902,153.450
C06708=1078.924,-71.228,-55.632,173.514,19.899,153.450
C06709=1078.918,-71.477,-55.621,173.512,19.898,153.450
C06710=1078.912,-71.728,-55.610,173.511,19.897,153.450
C06711=1078.907,-71.977,-55.598,173.509,19.895,153.450
C06712=1078.901,-72.227,-55.587,173.508,19.893,153.450
C06713=1078.895,-72.477,-55.576,173.506,19.892,153.450
C06714=1078.889,-72.727,-55.565,173.505,19.890,153.450
C06715=1078.883,-72.975,-55.554,173.503,19.889,153.450
C06716=1078.877,-73.226,-55.542,173.502,19.887,153.450
C06717=1078.871,-73.475,-55.531,173.501,19.885,153.450
C06718=1078.865,-73.725,-55.521,173.499,19.884,153.450
C06719=1078.859,-73.975,-55.509,173.498,19.882,153.450
C06720=1078.853,-74.224,-55.498,173.496,19.881,153.450
C06721=1078.847,-74.474,-55.488,173.495,19.879,153.450
C06722=1078.841,-74.724,-55.476,173.493,19.877,153.450
C06723=1078.835,-74.973,-55.465,173.492,19.876,153.450
C06724=1078.830,-75.223,-55.455,173.490,19.874,153.450
C06725=1078.823,-75.473,-55.443,173.488,19.872,153.450
C06726=1078.818,-75.723,-55.432,173.487,19.871,153.449
C06727=1078.812,-75.972,-55.422,173.485,19.869,153.449
C06728=1078.805,-76.222,-55.411,173.484,19.868,153.449
C06729=1078.799,-76.472,-55.400,173.482,19.866,153.449
C06730=1078.793,-76.721,-55.389,173.481,19.864,153.449
C06731=1078.787,-76.971,-55.378,173.479,19.863,153.449
C06732=1078.781,-77.221,-55.367,173.478,19.861,153.449
C06733=1078.775,-77.470,-55.356,173.476,19.860,153.449
C06734=1078.769,-77.720,-55.345,173.475,19.858,153.449
C06735=1078.763,-77.970,-55.334,173.473,19.857,153.449
C06736=1078.757,-78.219,-55.324,173.472,19.855,153.449
C06737=1078.751,-78.469,-55.313,173.470,19.854,153.449
C06738=1078.745,-78.719,-55.302,173.469,19.852,153.449
C06739=1078.739,-78.968,-55.291,173.467,19.851,153.449
C06740=1078.733,-79.218,-55.280,173.466,19.850,153.449
C06741=1078.727,-79.468,-55.269,173.465,19.848,153.449
C06742=1078.721,-79.718,-55.259,173.463,19.847,153.449
C06743=1078.715,-79.967,-55.248,173.462,19.845,153.449
C06744=1078.709,-80.217,-55.237,173.460,19.844,153.449
C06745=1078.703,-80.467,-55.226,173.459,19.842,153.449
C06746=1078.697,-80.716,-55.216,173.457,19.841,153.449
C06747=1078.691,-80.966,-55.205,173.456,19.839,153.449
C06748=1078.684,-81.244,-55.193,173.454,19.838,153.449
C06749=1078.676,-81.521,-55.181,173.453,19.836,153.449
C06750=1078.670,-81.799,-55.169,173.451,19.835,153.449
C06751=1078.663,-82.076,-55.157,173.449,19.833,153.449
C06752=1078.657,-82.326,-55.147,173.447,19.831,153.449
C06753=1078.651,-82.576,-55.136,173.446,19.830,153.449
C06754=1078.645,-82.826,-55.125,173.444,19.828,153.449
C06755=1078.638,-83.075,-55.115,173.444,19.827,153.449
C06756=1078.633,-83.325,-55.104,173.442,19.826,153.449
C06757=1078.627,-83.575,-55.094,173.441,19.824,153.449
C06758=1078.620,-83.825,-55.083,173.439,19.823,153.449
C06759=1078.614,-84.074,-55.072,173.438,19.821,153.449
C06760=1078.609,-84.324,-55.061,173.436,19.820,153.449
C06761=1078.602,-84.573,-55.051,173.434,19.819,153.449
C06762=1078.596,-84.824,-55.040,173.433,19.817,153.449
C06763=1078.590,-85.073,-55.030,173.432,19.816,153.449
C06764=1078.584,-85.322,-55.019,173.430,19.815,153.449
C06765=1078.578,-85.572,-55.008,173.429,19.813,153.449
C06766=1078.571,-85.822,-54.998,173.427,19.812,153.448
C06767=1078.566,-86.072,-54.988,173.426,19.810,153.448
C06768=1078.560,-86.321,-54.977,173.424,19.809,153.449
C06769=1078.553,-86.570,-54.966,173.422,19.808,153.449
C06770=1078.547,-86.821,-54.956,173.421,19.806,153.449
C06771=1078.542,-87.071,-54.945,173.419,19.805,153.448
C06772=1078.535,-87.320,-54.935,173.418,19.803,153.448
C06773=1078.529,-87.569,-54.924,173.416,19.802,153.448
C06774=1078.523,-87.820,-54.914,173.415,19.801,153.449
C06775=1078.517,-88.069,-54.903,173.413,19.799,153.449
C06776=1078.511,-88.319,-54.892,173.412,19.798,153.449
C06777=1078.505,-88.569,-54.883,173.410,19.796,153.448
C06778=1078.499,-88.818,-54.872,173.409,19.795,153.448
C06779=1078.493,-89.067,-54.861,173.407,19.793,153.448
C06780=1078.487,-89.318,-54.851,173.406,19.792,153.449
C06781=1078.480,-89.567,-54.841,173.404,19.791,153.449
C06782=1078.475,-89.817,-54.830,173.403,19.789,153.449
C06783=1078.469,-90.067,-54.820,173.401,19.788,153.448
C06784=1078.463,-90.316,-54.809,173.400,19.786,153.448
C06785=1078.457,-90.567,-54.799,173.398,19.786,153.449
C06786=1078.450,-90.816,-54.789,173.396,19.784,153.449
C06787=1078.444,-91.065,-54.778,173.395,19.783,153.449
C06788=1078.438,-91.315,-54.768,173.393,19.781,153.449
C06789=1078.432,-91.565,-54.757,173.392,19.780,153.449
C06790=1078.427,-91.815,-54.747,173.391,19.779,153.449
C06791=1078.421,-92.064,-54.737,173.390,19.778,153.449
C06792=1078.414,-92.314,-54.726,173.388,19.776,153.448
C06793=1078.408,-92.564,-54.716,173.386,19.775,153.449
C06794=1078.402,-92.814,-54.705,173.385,19.774,153.449
C06795=1078.396,-93.063,-54.696,173.383,19.772,153.449
C06796=1078.390,-93.313,-54.685,173.382,19.771,153.449
C06797=1078.384,-93.563,-54.675,173.380,19.770,153.449
C06798=1078.378,-93.812,-54.664,173.379,19.768,153.449
C06799=1078.372,-94.062,-54.655,173.377,19.767,153.449
C06800=1078.367,-94.311,-54.644,173.376,19.765,153.449
C06801=1078.361,-94.562,-54.633,173.374,19.764,153.449
C06802=1078.354,-94.811,-54.623,173.372,19.763,153.449
C06803=1078.349,-95.062,-54.613,173.371,19.761,153.449
C06804=1078.342,-95.311,-54.602,173.369,19.761,153.449
C06805=1078.337,-95.561,-54.592,173.368,19.759,153.449
C06806=1078.330,-95.810,-54.582,173.366,19.758,153.449
C06807=1078.325,-96.060,-54.572,173.365,19.756,153.449
C06808=1078.318,-96.309,-54.562,173.364,19.756,153.449
C06809=1078.313,-96.559,-54.551,173.362,19.754,153.449
C06810=1078.306,-96.809,-54.541,173.361,19.753,153.449
C06811=1078.301,-97.059,-54.531,173.359,19.752,153.449
C06812=1078.294,-97.339,-54.519,173.358,19.750,153.449
C06813=1078.287,-97.619,-54.508,173.355,19.748,153.449
C06814=1078.280,-97.899,-54.497,173.354,19.747,153.449
C06815=1078.273,-98.178,-54.485,173.352,19.746,153.449
C06816=1078.267,-98.428,-54.476,173.351,19.744,153.449
C06817=1078.262,-98.678,-54.466,173.349,19.743,153.449
C06818=1078.255,-98.927,-54.455,173.348,19.742,153.449
C06819=1078.248,-99.177,-54.445,173.346,19.741,153.449
C06820=1078.243,-99.427,-54.434,173.344,19.739,153.449
C06821=1078.236,-99.677,-54.425,173.343,19.739,153.449
C06822=1078.230,-99.927,-54.415,173.342,19.738,153.449
C06823=1078.224,-100.176,-54.404,173.340,19.737,153.449
C06824=1078.218,-100.426,-54.395,173.339,19.735,153.449
C06825=1078.212,-100.676,-54.385,173.337,19.734,153.449
C06826=1078.206,-100.925,-54.374,173.336,19.733,153.449
C06827=1078.200,-101.175,-54.365,173.334,19.732,153.449
C06828=1078.194,-101.425,-54.355,173.332,19.730,153.449
C06829=1078.188,-101.674,-54.345,173.331,19.729,153.450
C06830=1078.182,-101.924,-54.335,173.329,19.728,153.449
C06831=1078.176,-102.174,-54.325,173.327,19.727,153.450
C06832=1078.170,-102.423,-54.315,173.326,19.725,153.450
C06833=1078.164,-102.673,-54.305,173.325,19.725,153.450
C06834=1078.158,-102.923,-54.295,173.324,19.723,153.450
C06835=1078.151,-103.172,-54.285,173.322,19.722,153.450
C06836=1078.145,-103.422,-54.275,173.320,19.721,153.450
C06837=1078.139,-103.673,-54.265,173.319,19.720,153.450
C06838=1078.133,-103.922,-54.255,173.317,19.719,153.450
C06839=1078.127,-104.172,-54.245,173.315,19.718,153.450
C06840=1078.120,-104.421,-54.235,173.314,19.716,153.450
C06841=1078.115,-104.672,-54.225,173.312,19.715,153.450
C06842=1078.109,-104.921,-54.216,173.311,19.714,153.450
C06843=1078.102,-105.171,-54.205,173.310,19.713,153.450
C06844=1078.096,-105.420,-54.196,173.308,19.712,153.450
C06845=1078.091,-105.670,-54.186,173.307,19.711,153.450
C06846=1078.085,-105.920,-54.176,173.305,19.710,153.450
C06847=1078.078,-106.169,-54.166,173.303,19.709,153.450
C06848=1078.072,-106.419,-54.156,173.302,19.707,153.450
C06849=1078.066,-106.669,-54.147,173.300,19.706,153.450
C06850=1078.060,-106.919,-54.137,173.299,19.705,153.450
C06851=1078.054,-107.169,-54.127,173.297,19.704,153.451
C06852=1078.048,-107.418,-54.117,173.296,19.704,153.451
C06853=1078.042,-107.667,-54.108,173.295,19.702,153.451
C06854=1078.035,-107.918,-54.098,173.293,19.701,153.451
C06855=1078.029,-108.167,-54.088,173.291,19.700,153.451
C06856=1078.024,-108.418,-54.078,173.290,19.699,153.451
C06857=1078.018,-108.667,-54.069,173.288,19.698,153.451
C06858=1078.012,-108.916,-54.059,173.286,19.697,153.451
C06859=1078.005,-109.166,-54.049,173.285,19.695,153.451
C06860=1077.999,-109.415,-54.039,173.284,19.695,153.451
C06861=1077.993,-109.665,-54.030,173.282,19.694,153.451
C06862=1077.987,-109.915,-54.020,173.280,19.693,153.451
C06863=1077.981,-110.165,-54.011,173.279,19.692,153.451
C06864=1077.975,-110.415,-54.001,173.277,19.691,153.451
C06865=1077.968,-110.664,-53.991,173.275,19.690,153.452
C06866=1077.962,-110.914,-53.982,173.274,19.689,153.452
C06867=1077.956,-111.164,-53.972,173.272,19.687,153.452
C06868=1077.950,-111.414,-53.961,173.271,19.687,153.452
C06869=1077.944,-111.663,-53.952,173.270,19.686,153.452
C06870=1077.938,-111.913,-53.942,173.268,19.685,153.452
C06871=1077.932,-112.163,-53.933,173.266,19.683,153.452
C06872=1077.926,-112.413,-53.923,173.265,19.682,153.452
C06873=1077.919,-112.663,-53.914,173.263,19.681,153.452
C06874=1077.913,-112.912,-53.904,173.261,19.681,153.452
C06875=1077.907,-113.162,-53.894,173.260,19.679,153.452
C06876=1077.901,-113.439,-53.884,173.258,19.678,153.452
C06877=1077.894,-113.716,-53.873,173.256,19.677,153.452
C06878=1077.887,-113.993,-53.863,173.255,19.676,153.453
C06879=1077.880,-114.270,-53.853,173.253,19.675,153.453
C06880=1077.874,-114.520,-53.843,173.251,19.674,153.453
C06881=1077.868,-114.770,-53.833,173.251,19.673,153.453
C06882=1077.862,-115.019,-53.824,173.249,19.672,153.453
C06883=1077.856,-115.269,-53.814,173.247,19.671,153.453
C06884=1077.850,-115.519,-53.805,173.245,19.670,153.453
C06885=1077.843,-115.769,-53.795,173.244,19.670,153.453
C06886=1077.837,-116.019,-53.786,173.242,19.669,153.453
C06887=1077.831,-116.268,-53.776,173.241,19.667,153.453
C06888=1077.825,-116.518,-53.767,173.240,19.667,153.453
C06889=1077.819,-116.767,-53.757,173.238,19.666,153.454
C06890=1077.813,-117.017,-53.748,173.236,19.665,153.454
C06891=1077.807,-117.267,-53.738,173.235,19.664,153.454
C06892=1077.801,-117.517,-53.729,173.233,19.663,153.454
C06893=1077.795,-117.767,-53.719,173.231,19.662,153.454
C06894=1077.788,-118.016,-53.710,173.230,19.661,153.454
C06895=1077.782,-118.266,-53.701,173.229,19.660,153.454
C06896=1077.776,-118.516,-53.692,173.227,19.660,153.454
C06897=1077.770,-118.765,-53.682,173.225,19.659,153.454
C06898=1077.764,-119.015,-53.673,173.223,19.658,153.455
C06899=1077.758,-119.265,-53.663,173.222,19.657,153.455
C06900=1077.752,-119.515,-53.654,173.221,19.656,153.455
C06901=1077.745,-119.765,-53.644,173.219,19.655,153.455
C06902=1077.739,-120.014,-53.635,173.218,19.654,153.455
C06903=1077.733,-120.265,-53.626,173.216,19.653,153.455
C06904=1077.727,-120.514,-53.617,173.214,19.652,153.455
C06905=1077.721,-120.763,-53.608,173.212,19.651,153.455
C06906=1077.715,-121.013,-53.598,173.212,19.650,153.455
C06907=1077.709,-121.263,-53.588,173.210,19.650,153.455
C06908=1077.702,-121.513,-53.579,173.208,19.649,153.455
C06909=1077.697,-121.763,-53.570,173.206,19.648,153.456
C06910=1077.691,-122.012,-53.561,173.205,19.647,153.456
C06911=1077.684,-122.262,-53.552,173.203,19.646,153.456
C06912=1077.678,-122.512,-53.542,173.202,19.646,153.456
C06913=1077.672,-122.761,-53.533,173.200,19.645,153.456
C06914=1077.666,-123.012,-53.524,173.198,19.644,153.456
C06915=1077.660,-123.262,-53.514,173.197,19.643,153.456
C06916=1077.654,-123.511,-53.505,173.195,19.642,153.457
C06917=1077.647,-123.760,-53.496,173.194,19.642,153.457
C06918=1077.641,-124.010,-53.486,173.192,19.641,153.457
C06919=1077.635,-124.260,-53.478,173.191,19.640,153.457
C06920=1077.629,-124.510,-53.468,173.189,19.639,153.457
C06921=1077.623,-124.759,-53.459,173.187,19.638,153.457
C06922=1077.616,-125.009,-53.450,173.186,19.637,153.457
C06923=1077.611,-125.259,-53.441,173.185,19.636,153.457
C06924=1077.604,-125.509,-53.431,173.183,19.636,153.457
C06925=1077.598,-125.758,-53.423,173.181,19.635,153.458
C06926=1077.592,-126.009,-53.414,173.179,19.634,153.458
C06927=1077.586,-126.258,-53.404,173.178,19.633,153.458
C06928=1077.580,-126.508,-53.395,173.177,19.633,153.458
C06929=1077.573,-126.758,-53.387,173.175,19.632,153.458
C06930=1077.567,-127.008,-53.377,173.173,19.631,153.458
C06931=1077.561,-127.257,-53.367,173.171,19.630,153.458
C06932=1077.555,-127.508,-53.359,173.170,19.630,153.458
C06933=1077.548,-127.757,-53.350,173.169,19.629,153.459
C06934=1077.542,-128.008,-53.341,173.167,19.628,153.459
C06935=1077.539,-128.258,-53.331,173.166,19.627,153.459
C06936=1077.538,-128.513,-53.319,173.165,19.624,153.458
C06937=1077.540,-128.767,-53.307,173.164,19.621,153.458
C06938=1077.545,-129.020,-53.294,173.163,19.617,153.457
C06939=1077.552,-129.270,-53.280,173.164,19.611,153.456
C06940=1077.156,-129.292,-53.428,173.119,19.737,153.487
C06941=1077.148,-129.041,-53.443,173.119,19.743,153.488
C06942=1077.143,-128.789,-53.455,173.119,19.747,153.489
C06943=1077.141,-128.535,-53.468,173.120,19.750,153.489
C06944=1077.142,-128.280,-53.479,173.121,19.752,153.490
C06945=1077.145,-128.030,-53.489,173.122,19.754,153.490
C06946=1077.151,-127.779,-53.498,173.124,19.755,153.490
C06947=1077.157,-127.530,-53.508,173.126,19.756,153.489
C06948=1077.164,-127.279,-53.516,173.127,19.756,153.489
C06949=1077.170,-127.030,-53.526,173.128,19.757,153.489
C06950=1077.176,-126.780,-53.535,173.130,19.758,153.489
C06951=1077.182,-126.529,-53.544,173.132,19.759,153.489
C06952=1077.189,-126.280,-53.553,173.133,19.760,153.489
C06953=1077.195,-126.031,-53.562,173.134,19.760,153.489
C06954=1077.200,-125.780,-53.571,173.136,19.761,153.489
C06955=1077.207,-125.531,-53.581,173.138,19.762,153.488
C06956=1077.214,-125.281,-53.590,173.140,19.763,153.488
C06957=1077.220,-125.031,-53.599,173.141,19.764,153.488
C06958=1077.225,-124.782,-53.608,173.143,19.765,153.488
C06959=1077.232,-124.532,-53.617,173.144,19.765,153.488
C06960=1077.238,-124.282,-53.626,173.146,19.766,153.488
C06961=1077.244,-124.033,-53.636,173.147,19.767,153.488
C06962=1077.250,-123.782,-53.645,173.149,19.767,153.487
C06963=1077.256,-123.532,-53.654,173.151,19.768,153.487
C06964=1077.262,-123.283,-53.664,173.152,19.769,153.487
C06965=1077.269,-123.034,-53.672,173.154,19.770,153.487
C06966=1077.275,-122.783,-53.681,173.155,19.771,153.487
C06967=1077.281,-122.534,-53.691,173.157,19.772,153.487
C06968=1077.287,-122.284,-53.700,173.159,19.773,153.487
C06969=1077.293,-122.035,-53.710,173.161,19.773,153.487
C06970=1077.299,-121.785,-53.719,173.161,19.774,153.487
C06971=1077.305,-121.535,-53.727,173.163,19.775,153.487
C06972=1077.312,-121.285,-53.737,173.165,19.776,153.486
C06973=1077.318,-121.035,-53.747,173.167,19.777,153.486
C06974=1077.324,-120.785,-53.756,173.168,19.778,153.486
C06975=1077.330,-120.536,-53.766,173.170,19.779,153.486
C06976=1077.336,-120.286,-53.775,173.171,19.779,153.486
C06977=1077.341,-120.036,-53.784,173.173,19.780,153.486
C06978=1077.348,-119.787,-53.793,173.174,19.781,153.486
C06979=1077.355,-119.537,-53.802,173.176,19.782,153.486
C06980=1077.361,-119.287,-53.812,173.178,19.783,153.486
C06981=1077.367,-119.037,-53.821,173.179,19.784,153.486
C06982=1077.373,-118.787,-53.831,173.180,19.785,153.485
C06983=1077.379,-118.538,-53.840,173.182,19.786,153.485
C06984=1077.385,-118.288,-53.850,173.184,19.787,153.485
C06985=1077.391,-118.039,-53.859,173.185,19.788,153.485
C06986=1077.397,-117.788,-53.868,173.187,19.789,153.485
C06987=1077.403,-117.538,-53.878,173.189,19.790,153.485
C06988=1077.409,-117.289,-53.887,173.190,19.790,153.485
C06989=1077.416,-117.039,-53.896,173.191,19.791,153.485
C06990=1077.422,-116.789,-53.906,173.193,19.792,153.485
C06991=1077.428,-116.540,-53.915,173.195,19.793,153.485
C06992=1077.434,-116.290,-53.925,173.196,19.794,153.484
C06993=1077.440,-116.041,-53.934,173.198,19.795,153.484
C06994=1077.446,-115.791,-53.944,173.200,19.796,153.484
C06995=1077.453,-115.541,-53.953,173.201,19.797,153.484
C06996=1077.459,-115.291,-53.963,173.202,19.798,153.484
C06997=1077.465,-115.041,-53.973,173.204,19.799,153.484
C06998=1077.471,-114.792,-53.982,173.206,19.800,153.484
C06999=1077.477,-114.542,-53.992,173.207,19.801,153.484
C07000=1077.483,-114.292,-54.001,173.209,19.802,153.484
C07001=1077.490,-114.015,-54.012,173.211,19.803,153.484
C07002=1077.496,-113.738,-54.022,173.212,19.804,153.483
C07003=1077.503,-113.461,-54.033,173.214,19.805,153.484
C07004=1077.511,-113.183,-54.044,173.216,19.806,153.483
C07005=1077.517,-112.934,-54.053,173.217,19.807,153.483
C07006=1077.522,-112.683,-54.063,173.219,19.808,153.483
C07007=1077.528,-112.434,-54.073,173.221,19.810,153.483
C07008=1077.534,-112.185,-54.082,173.221,19.810,153.483
C07009=1077.540,-111.935,-54.092,173.223,19.811,153.483
C07010=1077.546,-111.685,-54.101,173.225,19.812,153.483
C07011=1077.553,-111.435,-54.111,173.226,19.813,153.483
C07012=1077.559,-111.185,-54.120,173.228,19.814,153.483
C07013=1077.565,-110.936,-54.130,173.230,19.815,153.483
C07014=1077.571,-110.686,-54.139,173.232,19.816,153.483
C07015=1077.578,-110.437,-54.150,173.233,19.818,153.483
C07016=1077.584,-110.187,-54.159,173.234,19.818,153.483
C07017=1077.590,-109.937,-54.169,173.236,19.819,153.482
C07018=1077.596,-109.687,-54.178,173.237,19.821,153.482
C07019=1077.602,-109.437,-54.189,173.239,19.821,153.482
C07020=1077.608,-109.187,-54.198,173.241,19.822,153.482
C07021=1077.614,-108.938,-54.208,173.242,19.824,153.482
C07022=1077.620,-108.688,-54.217,173.244,19.825,153.482
C07023=1077.627,-108.439,-54.228,173.245,19.826,153.482
C07024=1077.633,-108.189,-54.237,173.246,19.827,153.482
C07025=1077.639,-107.939,-54.247,173.248,19.828,153.482
C07026=1077.645,-107.689,-54.256,173.250,19.829,153.482
C07027=1077.651,-107.439,-54.266,173.251,19.830,153.482
C07028=1077.657,-107.189,-54.276,173.253,19.831,153.482
C07029=1077.663,-106.940,-54.286,173.254,19.832,153.482
C07030=1077.669,-106.690,-54.296,173.256,19.833,153.482
C07031=1077.675,-106.440,-54.305,173.258,19.834,153.482
C07032=1077.682,-106.191,-54.315,173.259,19.836,153.482
C07033=1077.687,-105.941,-54.325,173.260,19.836,153.481
C07034=1077.694,-105.691,-54.335,173.262,19.837,153.481
C07035=1077.700,-105.442,-54.345,173.263,19.839,153.481
C07036=1077.706,-105.192,-54.355,173.265,19.840,153.481
C07037=1077.711,-104.942,-54.365,173.266,19.841,153.481
C07038=1077.718,-104.692,-54.375,173.268,19.842,153.481
C07039=1077.724,-104.443,-54.385,173.270,19.844,153.481
C07040=1077.730,-104.193,-54.394,173.271,19.845,153.481
C07041=1077.736,-103.943,-54.404,173.273,19.846,153.481
C07042=1077.742,-103.694,-54.415,173.275,19.847,153.481
C07043=1077.748,-103.444,-54.424,173.276,19.848,153.481
C07044=1077.754,-103.194,-54.434,173.277,19.849,153.481
C07045=1077.760,-102.944,-54.444,173.278,19.850,153.481
C07046=1077.766,-102.695,-54.454,173.280,19.851,153.481
C07047=1077.772,-102.445,-54.464,173.282,19.853,153.481
C07048=1077.779,-102.195,-54.473,173.283,19.854,153.481
C07049=1077.784,-101.946,-54.484,173.285,19.855,153.481
C07050=1077.791,-101.696,-54.494,173.287,19.856,153.481
C07051=1077.797,-101.446,-54.503,173.288,19.858,153.481
C07052=1077.802,-101.197,-54.514,173.290,19.859,153.481
C07053=1077.809,-100.947,-54.524,173.291,19.860,153.481
C07054=1077.815,-100.697,-54.533,173.293,19.861,153.480
C07055=1077.822,-100.447,-54.544,173.294,19.862,153.481
C07056=1077.827,-100.197,-54.554,173.295,19.863,153.480
C07057=1077.833,-99.947,-54.564,173.297,19.864,153.480
C07058=1077.840,-99.698,-54.574,173.299,19.865,153.480
C07059=1077.845,-99.448,-54.584,173.300,19.867,153.480
C07060=1077.852,-99.199,-54.594,173.302,19.868,153.480
C07061=1077.858,-98.949,-54.604,173.303,19.869,153.480
C07062=1077.863,-98.699,-54.614,173.305,19.871,153.480
C07063=1077.870,-98.450,-54.624,173.307,19.872,153.480
C07064=1077.876,-98.200,-54.634,173.308,19.873,153.480
C07065=1077.883,-97.920,-54.646,173.310,19.875,153.480
C07066=1077.890,-97.639,-54.657,173.311,19.876,153.480
C07067=1077.896,-97.360,-54.669,173.313,19.877,153.480
C07068=1077.903,-97.079,-54.680,173.314,19.879,153.480
C07069=1077.910,-96.830,-54.690,173.316,19.879,153.480
C07070=1077.915,-96.580,-54.700,173.317,19.881,153.480
C07071=1077.922,-96.331,-54.711,173.319,19.882,153.480
C07072=1077.927,-96.080,-54.721,173.320,19.884,153.480
C07073=1077.934,-95.831,-54.731,173.322,19.885,153.480
C07074=1077.939,-95.581,-54.741,173.324,19.886,153.480
C07075=1077.945,-95.332,-54.752,173.325,19.888,153.480
C07076=1077.951,-95.082,-54.762,173.327,19.889,153.480
C07077=1077.957,-94.832,-54.773,173.328,19.890,153.480
C07078=1077.963,-94.583,-54.782,173.330,19.892,153.480
C07079=1077.969,-94.333,-54.793,173.331,19.893,153.480
C07080=1077.976,-94.083,-54.803,173.333,19.894,153.480
C07081=1077.981,-93.833,-54.814,173.335,19.896,153.480
C07082=1077.987,-93.583,-54.823,173.336,19.897,153.480
C07083=1077.993,-93.334,-54.834,173.338,19.899,153.480
C07084=1077.999,-93.084,-54.844,173.339,19.899,153.480
C07085=1078.005,-92.835,-54.855,173.341,19.901,153.480
C07086=1078.011,-92.585,-54.864,173.341,19.902,153.480
C07087=1078.017,-92.335,-54.875,173.343,19.903,153.480
C07088=1078.024,-92.086,-54.885,173.344,19.905,153.480
C07089=1078.030,-91.835,-54.896,173.346,19.906,153.480
C07090=1078.035,-91.586,-54.907,173.348,19.907,153.480
C07091=1078.041,-91.336,-54.916,173.349,19.909,153.480
C07092=1078.047,-91.086,-54.927,173.351,19.910,153.480
C07093=1078.054,-90.837,-54.938,173.352,19.912,153.480
C07094=1078.059,-90.587,-54.948,173.354,19.913,153.480
C07095=1078.066,-90.337,-54.958,173.355,19.914,153.480
C07096=1078.072,-90.087,-54.969,173.357,19.916,153.480
C07097=1078.077,-89.838,-54.979,173.358,19.917,153.480
C07098=1078.084,-89.589,-54.990,173.360,19.919,153.480
C07099=1078.089,-89.338,-55.000,173.361,19.920,153.480
C07100=1078.096,-89.089,-55.010,173.363,19.921,153.480
C07101=1078.102,-88.839,-55.021,173.364,19.922,153.480
C07102=1078.108,-88.589,-55.032,173.366,19.924,153.480
C07103=1078.114,-88.340,-55.042,173.367,19.925,153.480
C07104=1078.120,-88.090,-55.053,173.369,19.927,153.480
C07105=1078.126,-87.840,-55.062,173.371,19.928,153.480
C07106=1078.132,-87.590,-55.074,173.372,19.929,153.480
C07107=1078.139,-87.341,-55.084,173.374,19.931,153.480
C07108=1078.144,-87.092,-55.095,173.375,19.932,153.480
C07109=1078.150,-86.841,-55.105,173.377,19.934,153.480
C07110=1078.156,-86.592,-55.115,173.378,19.935,153.480
C07111=1078.163,-86.342,-55.126,173.380,19.937,153.480
C07112=1078.168,-86.092,-55.137,173.381,19.938,153.480
C07113=1078.175,-85.843,-55.147,173.383,19.939,153.480
C07114=1078.180,-85.593,-55.158,173.384,19.941,153.480
C07115=1078.187,-85.343,-55.168,173.386,19.942,153.480
C07116=1078.193,-85.093,-55.179,173.387,19.944,153.480
C07117=1078.199,-84.844,-55.189,173.389,19.945,153.480
C07118=1078.205,-84.595,-55.200,173.389,19.946,153.480
C07119=1078.211,-84.344,-55.211,173.391,19.947,153.480
C07120=1078.217,-84.095,-55.222,173.392,19.949,153.480
C07121=1078.223,-83.845,-55.231,173.394,19.950,153.480
C07122=1078.230,-83.595,-55.243,173.395,19.952,153.480
C07123=1078.235,-83.346,-55.253,173.397,19.953,153.480
C07124=1078.242,-83.096,-55.264,173.398,19.955,153.480
C07125=1078.248,-82.847,-55.275,173.400,19.956,153.480
C07126=1078.254,-82.596,-55.285,173.402,19.957,153.480
C07127=1078.260,-82.347,-55.295,173.403,19.959,153.480
C07128=1078.266,-82.097,-55.306,173.405,19.960,153.480
C07129=1078.272,-81.819,-55.318,173.407,19.962,153.480
C07130=1078.280,-81.542,-55.330,173.408,19.964,153.480
C07131=1078.287,-81.264,-55.342,173.410,19.965,153.480
C07132=1078.293,-80.986,-55.354,173.411,19.967,153.480
C07133=1078.300,-80.737,-55.364,173.413,19.969,153.480
C07134=1078.306,-80.486,-55.375,173.414,19.970,153.480
C07135=1078.312,-80.237,-55.386,173.416,19.971,153.480
C07136=1078.318,-79.987,-55.397,173.417,19.972,153.480
C07137=1078.325,-79.738,-55.408,173.419,19.974,153.480
C07138=1078.330,-79.488,-55.419,173.420,19.976,153.480
C07139=1078.336,-79.239,-55.430,173.422,19.977,153.481
C07140=1078.342,-78.989,-55.440,173.423,19.979,153.481
C07141=1078.348,-78.739,-55.452,173.425,19.980,153.481
C07142=1078.354,-78.489,-55.463,173.426,19.982,153.481
C07143=1078.360,-78.240,-55.473,173.428,19.983,153.481
C07144=1078.367,-77.990,-55.484,173.429,19.985,153.481
C07145=1078.372,-77.740,-55.494,173.431,19.986,153.481
C07146=1078.378,-77.490,-55.505,173.432,19.988,153.481
C07147=1078.384,-77.241,-55.516,173.434,19.989,153.481
C07148=1078.390,-76.991,-55.527,173.435,19.991,153.481
C07149=1078.396,-76.741,-55.538,173.436,19.993,153.481
C07150=1078.402,-76.492,-55.549,173.438,19.994,153.481
C07151=1078.409,-76.242,-55.560,173.439,19.996,153.481
C07152=1078.414,-75.992,-55.571,173.441,19.997,153.481
C07153=1078.420,-75.743,-55.581,173.442,19.999,153.481
C07154=1078.426,-75.493,-55.593,173.444,20.000,153.481
C07155=1078.432,-75.243,-55.604,173.445,20.002,153.481
C07156=1078.438,-74.994,-55.614,173.447,20.004,153.481
C07157=1078.445,-74.744,-55.626,173.449,20.006,153.481
C07158=1078.450,-74.495,-55.637,173.451,20.007,153.481
C07159=1078.457,-74.245,-55.649,173.452,20.008,153.481
C07160=1078.462,-73.995,-55.659,173.454,20.010,153.481
C07161=1078.468,-73.746,-55.670,173.455,20.012,153.481
C07162=1078.474,-73.495,-55.682,173.456,20.013,153.481
C07163=1078.480,-73.246,-55.692,173.458,20.015,153.481
C07164=1078.486,-72.996,-55.703,173.459,20.016,153.481
C07165=1078.492,-72.747,-55.714,173.461,20.018,153.482
C07166=1078.498,-72.497,-55.725,173.462,20.020,153.482
C07167=1078.504,-72.247,-55.736,173.464,20.021,153.482
C07168=1078.509,-71.998,-55.747,173.465,20.023,153.482
C07169=1078.516,-71.748,-55.759,173.466,20.025,153.482
C07170=1078.522,-71.499,-55.770,173.468,20.026,153.482
C07171=1078.527,-71.249,-55.781,173.469,20.028,153.482
C07172=1078.533,-70.999,-55.793,173.471,20.030,153.482
C07173=1078.539,-70.749,-55.804,173.472,20.031,153.482
C07174=1078.545,-70.500,-55.814,173.474,20.033,153.482
C07175=1078.551,-70.250,-55.826,173.475,20.035,153.482
C07176=1078.557,-70.001,-55.837,173.476,20.036,153.482
C07177=1078.563,-69.750,-55.849,173.478,20.038,153.482
C07178=1078.569,-69.501,-55.859,173.479,20.040,153.483
C07179=1078.574,-69.251,-55.871,173.481,20.041,153.483
C07180=1078.581,-69.001,-55.882,173.482,20.043,153.483
C07181=1078.587,-68.752,-55.894,173.483,20.045,153.483
C07182=1078.592,-68.503,-55.905,173.485,20.046,153.483
C07183=1078.599,-68.252,-55.916,173.486,20.048,153.483
C07184=1078.604,-68.003,-55.927,173.488,20.050,153.483
C07185=1078.611,-67.753,-55.938,173.490,20.052,153.483
C07186=1078.616,-67.504,-55.950,173.491,20.053,153.483
C07187=1078.622,-67.254,-55.961,173.493,20.055,153.483
C07188=1078.628,-67.004,-55.972,173.494,20.056,153.483
C07189=1078.634,-66.754,-55.983,173.496,20.058,153.483
C07190=1078.640,-66.505,-55.995,173.497,20.060,153.483
C07191=1078.646,-66.255,-56.006,173.499,20.061,153.483
C07192=1078.651,-66.006,-56.017,173.500,20.063,153.484
C07193=1078.658,-65.730,-56.030,173.501,20.065,153.484
C07194=1078.665,-65.454,-56.043,173.503,20.067,153.484
C07195=1078.671,-65.179,-56.054,173.505,20.069,153.484
C07196=1078.678,-64.904,-56.068,173.506,20.071,153.484
C07197=1078.685,-64.653,-56.079,173.508,20.072,153.484
C07198=1078.690,-64.404,-56.090,173.509,20.074,153.484
C07199=1078.696,-64.154,-56.103,173.510,20.076,153.484
C07200=1078.702,-63.905,-56.113,173.512,20.077,153.484
C07201=1078.708,-63.655,-56.124,173.513,20.079,153.484
C07202=1078.714,-63.405,-56.136,173.515,20.081,153.484
C07203=1078.720,-63.156,-56.147,173.516,20.082,153.484
C07204=1078.726,-62.905,-56.159,173.517,20.084,153.485
C07205=1078.732,-62.657,-56.171,173.520,20.086,153.484
C07206=1078.738,-62.406,-56.182,173.521,20.088,153.485
C07207=1078.744,-62.157,-56.193,173.523,20.090,153.485
C07208=1078.750,-61.907,-56.205,173.524,20.091,153.485
C07209=1078.755,-61.658,-56.216,173.525,20.093,153.485
C07210=1078.762,-61.408,-56.228,173.527,20.095,153.485
C07211=1078.768,-61.158,-56.239,173.528,20.097,153.485
C07212=1078.774,-60.909,-56.251,173.530,20.098,153.485
C07213=1078.779,-60.659,-56.262,173.531,20.100,153.485
C07214=1078.786,-60.409,-56.274,173.532,20.102,153.485
C07215=1078.792,-60.160,-56.285,173.534,20.104,153.485
C07216=1078.798,-59.910,-56.297,173.535,20.105,153.485
C07217=1078.805,-59.660,-56.309,173.537,20.107,153.486
C07218=1078.810,-59.410,-56.320,173.538,20.109,153.486
C07219=1078.817,-59.161,-56.332,173.539,20.110,153.486
C07220=1078.822,-58.911,-56.343,173.542,20.112,153.486
C07221=1078.829,-58.662,-56.355,173.543,20.114,153.486
C07222=1078.834,-58.412,-56.366,173.544,20.116,153.486
C07223=1078.841,-58.162,-56.378,173.546,20.117,153.486
C07224=1078.846,-57.913,-56.389,173.547,20.119,153.486
C07225=1078.852,-57.663,-56.402,173.549,20.121,153.486
C07226=1078.859,-57.413,-56.413,173.550,20.123,153.486
C07227=1078.865,-57.164,-56.424,173.551,20.124,153.486
C07228=1078.871,-56.914,-56.436,173.553,20.126,153.487
C07229=1078.876,-56.665,-56.448,173.554,20.128,153.487
C07230=1078.883,-56.414,-56.459,173.555,20.130,153.487
C07231=1078.889,-56.165,-56.471,173.557,20.131,153.487
C07232=1078.895,-55.916,-56.483,173.559,20.134,153.487
C07233=1078.901,-55.666,-56.495,173.561,20.135,153.487
C07234=1078.907,-55.417,-56.506,173.562,20.137,153.487
C07235=1078.913,-55.166,-56.517,173.563,20.139,153.487
C07236=1078.919,-54.917,-56.530,173.565,20.141,153.487
C07237=1078.925,-54.667,-56.541,173.566,20.142,153.487
C07238=1078.932,-54.418,-56.553,173.567,20.144,153.488
C07239=1078.937,-54.168,-56.565,173.569,20.146,153.488
C07240=1078.943,-53.918,-56.576,173.570,20.148,153.488
C07241=1078.950,-53.669,-56.588,173.572,20.149,153.488
C07242=1078.955,-53.419,-56.600,173.573,20.151,153.488
C07243=1078.961,-53.169,-56.612,173.574,20.153,153.488
C07244=1078.968,-52.920,-56.624,173.577,20.155,153.488
C07245=1078.973,-52.670,-56.636,173.578,20.157,153.488
C07246=1078.980,-52.420,-56.647,173.579,20.159,153.488
C07247=1078.986,-52.171,-56.659,173.581,20.160,153.488
C07248=1078.992,-51.922,-56.671,173.582,20.162,153.488
C07249=1078.998,-51.671,-56.682,173.584,20.163,153.488
C07250=1079.005,-51.422,-56.694,173.585,20.165,153.489
C07251=1079.010,-51.173,-56.707,173.586,20.167,153.489
C07252=1079.016,-50.922,-56.718,173.588,20.169,153.489
C07253=1079.023,-50.673,-56.730,173.589,20.170,153.489
C07254=1079.029,-50.423,-56.742,173.591,20.173,153.489
C07255=1079.035,-50.174,-56.754,173.593,20.175,153.489
C07256=1079.041,-49.924,-56.766,173.594,20.176,153.489
C07257=1079.048,-49.650,-56.779,173.595,20.178,153.489
C07258=1079.054,-49.375,-56.792,173.597,20.180,153.489
C07259=1079.060,-49.101,-56.805,173.599,20.183,153.490
C07260=1079.067,-48.828,-56.818,173.600,20.185,153.490
C07261=1079.072,-48.577,-56.830,173.601,20.187,153.490
C07262=1079.079,-48.328,-56.842,173.603,20.188,153.490
C07263=1079.084,-48.078,-56.854,173.604,20.190,153.490
C07264=1079.090,-47.828,-56.867,173.605,20.192,153.490
C07265=1079.097,-47.578,-56.878,173.608,20.194,153.490
C07266=1079.102,-47.329,-56.890,173.609,20.196,153.490
C07267=1079.108,-47.079,-56.903,173.610,20.198,153.491
C07268=1079.114,-46.830,-56.915,173.612,20.200,153.491
C07269=1079.120,-46.580,-56.927,173.613,20.202,153.491
